# B&R Automation Studio project LW_CapProcess
Automation Studio 4.9

## Configuration Config2

CPU PC_any, AutomationRuntime B4.91, Build 4.1.2, Safety 0.0, Vc V4.73.0

### Task classes (Cpu.sw)
```
Cyclic#1 (cycle 10000 us):
  AlarmsX <- AlarmsPkg.AlarmsX.prg
  CapPush <- CapPushPkg.CapPush.prg
  PickupArm <- PickupArmPkg.PickupArm.prg
  LogoCOnv <- LogoConvPkg.LogoCOnv.prg
  ClrDetect <- ClrDetectPkg.ClrDetect.prg
  LineGates <- LaneGatesPkg.LineGates.prg
  AutoCtrl <- AutoCtrlPkg.AutoCtrl.prg
  SortConv <- SortConvPkg.SortConv.prg
  ComTotal_P <- Libraries.ComTotal.ComTotal_P.prg
DataObjects: Acp10sys
NcDataObjects: acp10etxen <- acp10etxen.dob, gAxis01a <- gAxis01obj.gAxis01a.dob, gAxis01i <- gAxis01obj.gAxis01i.dob, gAxis02a <- gAxis02obj.gAxis02a.dob, gAxis02i <- gAxis02obj.gAxis02i.dob
Binaries: udbdef, mvLoader, arflatprv, TCData, TCLang, arsvcreg, FWRules, arcoal, acp10cfg, Acp10map, iomap, asfw, UserMgt, Alarms, Role, ashwac, sysconf, arconfig, TC, ashwd, User, LogoAxis, Axis01
Libraries: Acp10man, Acp10par, NcGlobal, Acp10sim, Acp10_MC, sys_lib, brsystem, runtime, MpAlarmX, MpBase, astime, MpAxis, MpCom, MpServer, MpUserX, operator, ComTotal_L, AsTCP, standard, ArEventLog, AsBrStr, asieccon, fileio, arcert, dataobj, aseth, ashw, aruser, arssl, powerlnk
```

### Hardware
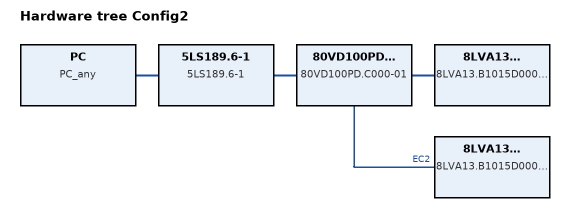
```
5LS189.6-1 : 5LS189.6-1 v1.5.0.0  [SL -> PC.SL1]
80VD100PD.C000-01 : 80VD100PD.C000-01 v2.5.0.0  [PLK1 -> 5LS189.6-1.IF2 (NodeNumber=1) [Cable Type=PowerlinkCable, Length=10, Version=1.0.0.3]; EC1 -> 8LVA13.B1015D000-0.EC; EC2 -> 8LVA13.B1015D000-0a.EC; MT2 -> 8LVA13.B1015D000-0a.MT]
  MotionTP = Acp10Arnc0
  Simulate = standard
  ActiveMotorSimulation_r1 = on
  BothEndSwitchesAreNormallyOpen_r1 = on
  ActiveMotorSimulation_r2 = on
  BothEndSwitchesAreNormallyOpen_r2 = on
8LVA13.B1015D000-0 : 8LVA13.B1015D000-0 v2.2.0.3  [EC -> 80VD100PD.C000-01.EC1; MT -> 80VD100PD.C000-01.MT1]
8LVA13.B1015D000-0a : 8LVA13.B1015D000-0 v2.2.0.3  [EC -> 80VD100PD.C000-01.EC2; MT -> 80VD100PD.C000-01.MT2]
PC : PC_any v1.1.1.0 (OrderNumber=PC)
  ConfigurationID = CapProcess_Config1
  Cyclic1Duration = 10000
  FileDevice1
  FileDeviceName1 = USER
  FileDevicePath1 = USER_PATH
  ActivateOpcUa = 1
  OpcUaInformationModels_PV_Version = 1
```

### Acp10cfg.ncc - PC/Motion/Acp10cfg.ncc
```
NcConfiguration (Version=5.23.1, NcSwId=Acp10)
  ACP10CF1_typ:
    cnt_nettrc_rec_drive = 1500
    bufsize_trace_upload = 1200
    tc_nc_man_task = Cyclic #1
    glob_pv_as_ncobject = Yes
    ncsys_dl_broadcast = Yes
    ncsys_dl_acp_reset = Yes
    safemc_log_err_to_ax = Yes
    network_init:
      ncsw_init_execute = Yes
      automatic_execute = No
      node_nr_warning = Yes
      net_err_before_ncact = Yes
    nettrc:
      enter_parsecrec = Yes
      enter_ncaction = Yes
      save_ring_startidx = Yes
    cam_prof_download:
      cam_dat_dl_parallel = No
      tc_cam_dl_parallel = Task class for NC Manager task
    plk_if[0]:
      if_name = SL1.IF2
      tc_CycDat_PLCopen = Task class for NC Manager task
      mc_broadcast_extdat = No
```

### Acp10map.ncm - PC/Motion/Acp10map.ncm
```
NcMapping (NcSwId=Acp10, DisabledNodesAreHidden=False)
  NcObject gAxis01 (ModuleId=80VD100PD.C000-01, Type=ncAXIS, Channel=1, AcoposSimulation=Standard, InitParameter=gAxis01i, AcoposParameter=gAxis01a, Disabled=FALSE, ModuleDisabled=FALSE)
  NcObject gAxis02 (ModuleId=80VD100PD.C000-01, Type=ncAXIS, Channel=2, AcoposSimulation=Standard, InitParameter=gAxis02i, AcoposParameter=gAxis02a, Disabled=FALSE, ModuleDisabled=FALSE)
  NcObject 80VD100PD.C000-01_ncV_AXIS1 (ModuleId=80VD100PD.C000-01, Type=ncV_AXIS, Channel=1, Disabled=TRUE, ModuleDisabled=FALSE)
  NcObject 80VD100PD.C000-01_ncV_AXIS2 (ModuleId=80VD100PD.C000-01, Type=ncV_AXIS, Channel=2, Disabled=TRUE, ModuleDisabled=FALSE)
```

### LogoAxis.mpaxisbasic - PC/Motion/LogoAxis.mpaxisbasic
```
Element gAxisBasic (Type=mpaxisbasic)
  Alarms = MpAlarmX
```

### SortAxis.mpaxisbasic - PC/Motion/SortAxis.mpaxisbasic
```
Element gAxisBasic_1 (Type=mpaxisbasic)
```

### PvMap.vvm - PC/PvMap.vvm
```iecst
VAR_CONFIG
	::ComTotal_SimInputs.CapPusher_LBK AT %Q.::CapPush:iCapPush.DIs.PusherLBK; (*Insert your comment here...*)
	::ComTotal_SimInputs.LogoAxis_ACTPOS AT %Q.::LogoCOnv:iLogoConv.DIs.LogoActPos; (*Insert your comment here...*)
	::ComTotal_SimInputs.CapPusher_LFR AT %Q.::CapPush:iCapPush.DIs.PusherLFR; (*Insert your comment here...*)
	::ComTotal_SimInputs.MagazineEmpty_IR AT %Q.::CapPush:iCapPush.DIs.MagznPosnEmpty_IR; (*Insert your comment here...*)
	::ComTotal_SimInputs.CapAtPickup_IR AT %Q.::CapPush:iCapPush.DIs.PickUp_IR; (*Insert your comment here...*)
	::ComTotal_SimInputs.ColourDetection_IR AT %Q.::ClrDetect:iClrDetect.DIs.ColorDetectionIR; (*Insert your comment here...*)
	::ComTotal_SimInputs.CapColour_NOT_BLACK AT %Q.::ClrDetect:iClrDetect.DIs.ColorDtectNotBlack; (*Insert your comment here...*)
	::ComTotal_SimInputs.CapColour_METALLIC AT %Q.::ClrDetect:iClrDetect.DIs.ColorDtectMetallic; (*Insert your comment here...*)
	::ComTotal_SimInputs.SortingConveyorStart_IR AT %Q.::SortConv:iSortConv.DIs.SortBasicConvStart_IR; (*Insert your comment here...*)
	::ComTotal_SimInputs.LogoConveyorStart_IR AT %Q.::LogoCOnv:iLogoConv.DIs.LogoConvStart_IR; (*Insert your comment here...*)
	::ComTotal_SimInputs.LogoConveyorExit_IR AT %Q.::LogoCOnv:iLogoConv.DIs.LogoConvExit_IR; (*Insert your comment here...*)
	::ComTotal_SimInputs.LaneGate1_LBK AT %Q.::LineGates:iLineGates.DIs.LG1_LBK; (*Insert your comment here...*)
	::ComTotal_SimInputs.LaneGate1_LFR AT %Q.::LineGates:iLineGates.DIs.LG1_LFR; (*Insert your comment here...*)
	::ComTotal_SimInputs.LaneGate2_LBK AT %Q.::LineGates:iLineGates.DIs.LG2_LBK; (*Insert your comment here...*)
	::ComTotal_SimInputs.LaneGate2_LFR AT %Q.::LineGates:iLineGates.DIs.LG2_LFR; (*Insert your comment here...*)
	::ComTotal_SimInputs.PickupArm_LBK AT %Q.::PickupArm:iPickupArm.DOs.PArmLBK; (*Insert your comment here...*)
	::ComTotal_SimInputs.PickupArm_LFR AT %Q.::PickupArm:iPickupArm.DOs.PArmLFR; (*Insert your comment here...*)
	::ComTotal_SimInputs.CapGripper_VACUUM AT %Q.::PickupArm:iPickupArm.DOs.CapGripVaccum; (*Insert your comment here...*)
	::ComTotal_SimInputs.LaneTop_IR AT %Q.::LineGates:iLineGates.DIs.LaneTopIR; (*Insert your comment here...*)
	::CapPush:iCapPush.DOs.PushFWD AT %Q.::ComTotal_SimOutputs.CapPusher_FWD; (*Insert your comment here...*)
	::SortConv:iSortConv.AOs.SortBasicConvSpeed AT %Q.::ComTotal_SimOutputs.SortingConveyor_SETSPEED; (*Insert your comment here...*)
	::LogoCOnv:iLogoConv.AOs.LogoConvSpeed AT %Q.::ComTotal_SimOutputs.LogoConveyor_SETSPEED; (*Insert your comment here...*)
	::LineGates:iLineGates.DOs.LG1FWD AT %Q.::ComTotal_SimOutputs.LaneGate1_FWD; (*Insert your comment here...*)
	::LineGates:iLineGates.DOs.LW2FWD AT %Q.::ComTotal_SimOutputs.LaneGate2_FWD; (*Insert your comment here...*)
	::PickupArm:iPickupArm.DIs.PArm_FWD AT %Q.::ComTotal_SimOutputs.PickupArm_FWD; (*Insert your comment here...*)
	::PickupArm:iPickupArm.DIs.PArm_BWD AT %Q.::ComTotal_SimOutputs.PickupArm_BWD; (*Insert your comment here...*)
	::PickupArm:iPickupArm.DIs.CapGripper_PICK AT %Q.::ComTotal_SimOutputs.CapGripper_PICK; (*Insert your comment here...*)
	::ClrDetect:iClrDetect.DOs.CapStopperFWD AT %Q.::ComTotal_SimOutputs.CapStopper_FWD; (*Insert your comment here...*)
END_VAR
```

### Alarms.mpalarmxcore - PC/mappServices/Alarms.mpalarmxcore
```
Element gAlarmXCore (Type=mpalarmxcore)
  mapp.AlarmX.Core:
    BySeverity:
      [0]:
        Severity = 50
        [0] = Reaction
          Name = Warning
      [1]:
        Severity = 100
        [0] = Reaction
          Name = EStop
  mapp.AlarmX.Core.Configuration:
    [0]:
      Name = CapPush
      Message = Magzine for cap is empty
      Severity = 10
      Behavior = PersistentAlarm
    [1]:
      Name = PArmError
      Message = Both Arms are on please disable one of it
      Severity = 100
      Behavior = PersistentAlarm
    [2]:
      Name = VaccumError
      Message = Arm is forward but no cap available to pick\
      Severity = 50
      Behavior = PersistentAlarm
    [3]:
      Name = ConvLogoErr
      Message = Cap is on the belt but velocity is zero
      Severity = 100
      Behavior = PersistentAlarm
    [4]:
      Name = ConvSortErr
      Message = Cap is on the belt but velocity is zero
      Severity = 100
      Behavior = PersistentAlarm
    [5]:
      Name = EStopCD
      Message = Estop for Color detect is pressed
      Severity = 100
      Behavior = PersistentAlarm
    [6]:
      Name = CapsFull
      Message = Maximum no of caps are filled please remove
      Severity = 100
      Behavior = PersistentAlarm
    [7]:
      Name = EStopLG
      Message = Emergency stop for line gate
      Severity = 100
      Behavior = PersistentAlarm
    [8]:
      Name = EStopAC
      Message = Emergency stop for main control has been pressed
      Severity = 100
      Behavior = PersistentAlarm
    [9]:
      Name = EStopAuto
      Message = Emergency stop is pressed
      Severity = 100
      Behavior = PersistentAlarm
Element gAlarmXCore_1 (Type=mpalarmxcore)
Element gAlarmXCore_2 (Type=mpalarmxcore)
```

### UserMgt.mpuserx - PC/mappServices/UserMgt.mpuserx
```
Element UserMgmtX (Type=mpuserx)
  ServerSettings:
    Server:
      AdditionalUserData:
        [0] = mail
        [1] = telephoneNumber
  Users:
    DefUser#1:
      id = admin
      lang = en
    DefUser#2:
      id = Anonymous
      lang = en
    DefUser#3:
      id = admin1
      lang = en
    DefUser#4:
      id = dev
      lang = en
    DefUser#5:
      id = yadnesh
      lang = en
  Groups:
    DefGroup#1:
      id = Administrators
      level = 100
      admin = TRUE
    DefGroup#2:
      id = Everyone
      admin = TRUE
    DefGroup#3:
      id = Operator
      level = 80
    DefGroup#4:
      id = Service
      level = 50
```

## Logical view

Binary libraries used (declarations not repeated): operator, runtime, astime, AsIecCon, Acp10man, Acp10par, NcGlobal, Acp10sim 5.23.1, Acp10_MC, sys_lib, brsystem, MpAlarmX, MpBase, MpAxis, MpCom, MpServer, MpUserX, AsTCP, standard, ArEventLog, AsBrStr

### Global.typ - Global data types
```iecst
TYPE
	gMainCmd_Str : 	STRUCT
		Stop : BOOL;
		EStop : BOOL;
		ErrorReset : BOOL;
		Start : BOOL;
	END_STRUCT;
END_TYPE
```

### Global.var - Global variables
```iecst
VAR
	gManuelMode : BOOL;
	gMainCmd : gMainCmd_Str;
	gAxis01 : ACP10AXIS_typ;
	gAxis02 : ACP10AXIS_typ;
	gColorCap : WSTRING[80];
END_VAR
```

### Package Logical/Libraries - Global libraries

### Package Logical/Libraries/ComTotal - Library package for ComTCP

### Library Logical/Libraries/ComTotal/ComTotal_L (ANSIC)

#### MNG_ComHdlr.hpp
```cpp
#ifndef _MNGCOMHDLR_HPP_
#define _MNGCOMHDLR_HPP_

#define TRUE  1
#define FALSE 0

#include "MNG_InternalTyp.hpp"

#include <bur/plc.h>
#include <bur/plctypes.h>
#include <AsTCP.h>
#include <standard.h>
#include <astime.h>
#include <runtime.h>
#include <AsBrStr.h>

typedef struct{
	TcpOpen_typ tcpOpen;
	TcpIoctl_typ tcpIoctl;
	tcpLINGER_typ tcpLINGER;
	TcpSend_typ tcpSend;
	TcpClose_typ tcpClose;
	TcpRecv_typ tcpRecv;
	TcpClient_typ tcpClient;
} asTcpFcn_t;

typedef enum {
	MNG_wSock,
	MNG_skippedMessage
} MNG_errorCases;

typedef enum {
	MNG_Init,
	MNG_Socket,
	MNG_Open,
	MNG_SetIo,
	MNG_Linger,
	MNG_Connecting,
	MNG_Exchange,
	MNG_Closing,
        MNG_Reset
} MNG_internalState_t;

	extern unsigned long int MNG_CpyOutToMsg(MNG_RawDatagram * pToServer, unsigned long int counter, ComTotal_OUTPUTS_32BIT_FWRD *pSimOutputs);
	extern unsigned long int MNG_CpyMsgToInp(MNG_RawDatagram * pFromServer, ComTotal_INPUTS_32BIT_FWRD *pSimInputs);

class MNG_ComHdlr
{
	public:

	MNG_ComHdlr(char *srvIpAdr, unsigned int srvPort, TIME sendCycleTime);
	~MNG_ComHdlr();

        int RunCommunication(void*, void*, BOOL*);

	private:

	char* _srvIpAdr;
	unsigned int _srvPort;
	TIME _sendCycleTime;

	unsigned int _error;

	MNG_internalState_t _internalState;
	TON_typ _connectionTon;
	TIME _connectionTime;

	bool _connect;
	bool _sendDone;

	signed int _recvOffset;

	signed long int _potMsgLen;
	signed long int _totalRecvLen;

	unsigned long int _one;
	unsigned long int _counter;
	unsigned long int _recvLen;
	unsigned long int _recvBuffer[10000];
	TON_typ _sendTon;
	MNG_RawDatagram _recvMessage;
	MNG_RawDatagram _sendMessage;

	static const signed long int SIXTEEN = 16;
	static const unsigned int PORT = 0;
	static const unsigned long int MNG_MAXPAYLOAD = 1400;

	void init_TcpOpen();
	void init_TcpSocket();
	void init_TcpIoctl();
	void init_TcpLinger();
	void init_TcpClient();
	void init_TcpRecv();
	void init_TcpSend(ComTotal_OUTPUTS_32BIT_FWRD* pSimOut);

	void InitParams();

	void SetSendDone(bool toogle);
	void SetStateValue(MNG_internalState_t stateVal);

};
#endif
```

#### MNG_Global.hpp
```cpp
#ifndef  _MNGGLOBAL_HPP_
#define _MNGGLOBAL_HPP_

#include <mng_globalTYP.h>

    typedef struct {

		signed short NumSignals;

        /* BOOL CapPusher_LBK */
        BOOL CapPusher_LBK;
        /* BOOL CapPusher_LFR */
        BOOL CapPusher_LFR;
        /* BOOL MagazineEmpty_IR */
        BOOL MagazineEmpty_IR;
        /* BOOL CapAtPickup_IR */
        BOOL CapAtPickup_IR;
        /* BOOL ColourDetection_IR */
        BOOL ColourDetection_IR;
        /* BOOL CapColour_NOT_BLACK */
        BOOL CapColour_NOT_BLACK;
        /* BOOL CapColour_METALLIC */
        BOOL CapColour_METALLIC;
        /* BOOL SortingConveyorStart_IR */
        BOOL SortingConveyorStart_IR;
        /* BOOL LogoConveyorStart_IR */
        BOOL LogoConveyorStart_IR;
        /* BOOL LogoConveyorExit_IR */
        BOOL LogoConveyorExit_IR;
        /* BOOL LaneGate1_LBK */
        BOOL LaneGate1_LBK;
        /* BOOL LaneGate1_LFR */
        BOOL LaneGate1_LFR;
        /* BOOL LaneGate2_LBK */
        BOOL LaneGate2_LBK;
        /* BOOL LaneGate2_LFR */
        BOOL LaneGate2_LFR;
        /* BOOL PickupArm_LBK */
        BOOL PickupArm_LBK;
        /* BOOL PickupArm_LFR */
        BOOL PickupArm_LFR;
        /* BOOL CapGripper_VACUUM */
        BOOL CapGripper_VACUUM;
        /* BOOL LaneTop_IR */
        BOOL LaneTop_IR;
        /* REAL LogoAxis_ACTPOS */
        REAL LogoAxis_ACTPOS;
        /* BOOL LogoStamper_LBK */
        BOOL LogoStamper_LBK;
        /* BOOL LogoStamper_LFR */
        BOOL LogoStamper_LFR;
        /* REAL PuncherAxis_ACTPOS */
        REAL PuncherAxis_ACTPOS;
        /* BOOL HolePuncher_LBK */
        BOOL HolePuncher_LBK;
        /* BOOL HolePuncher_LFR */
        BOOL HolePuncher_LFR;

        } ComTotal_INPUTS_32BIT_FWRD;

    typedef struct {

		signed short NumSignals;

        /* BOOL CapPusher_FWD */
        BOOL CapPusher_FWD;
        /* REAL SortingConveyor_SETSPEED */
        REAL SortingConveyor_SETSPEED;
        /* BOOL SortingConveyor_CLEAR */
        BOOL SortingConveyor_CLEAR;
        /* REAL LogoConveyor_SETSPEED */
        REAL LogoConveyor_SETSPEED;
        /* BOOL LogoConveyor_CLEAR */
        BOOL LogoConveyor_CLEAR;
        /* BOOL LaneGate1_FWD */
        BOOL LaneGate1_FWD;
        /* BOOL LaneGate2_FWD */
        BOOL LaneGate2_FWD;
        /* BOOL LaneStopper1_CLEAR */
        BOOL LaneStopper1_CLEAR;
        /* BOOL LaneStopper2_CLEAR */
        BOOL LaneStopper2_CLEAR;
        /* BOOL LaneStopper3_CLEAR */
        BOOL LaneStopper3_CLEAR;
        /* BOOL PickupArm_FWD */
        BOOL PickupArm_FWD;
        /* BOOL PickupArm_BWD */
        BOOL PickupArm_BWD;
        /* BOOL CapGripper_PICK */
        BOOL CapGripper_PICK;
        /* BOOL CapStopper_FWD */
        BOOL CapStopper_FWD;
        /* BOOL CP1586_PRESS */
        BOOL CP1586_PRESS;
        /* REAL LogoAxis_SETPOS */
        REAL LogoAxis_SETPOS;
        /* BOOL LogoStamper_FWD */
        BOOL LogoStamper_FWD;
        /* REAL PuncherAxis_SETPOS */
        REAL PuncherAxis_SETPOS;
        /* BOOL HolePuncher_FWD */
        BOOL HolePuncher_FWD;

        } ComTotal_OUTPUTS_32BIT_FWRD;

#endif
```

#### MNG_ComHdlr.cpp
```cpp
#include "MNG_ComHdlr.hpp"
#include "MNG_CpyMsgToInp.cpp"
#include "MNG_CpyOutToMsg.cpp"

asTcpFcn_t _asTcpFcn;

MNG_ComHdlr::MNG_ComHdlr(char *srvIpAdr, unsigned int srvPort, TIME sendCycleTime)
{
	_srvIpAdr = srvIpAdr;
	_srvPort = srvPort;
	_sendCycleTime = sendCycleTime;
	InitParams();
}

MNG_ComHdlr::~MNG_ComHdlr()
{
}

int MNG_ComHdlr::RunCommunication(void* pSimInputs, void* pSimOutputs, BOOL* pSimActive) {

        unsigned long int _lastCounter = _counter;

	ComTotal_INPUTS_32BIT_FWRD* pFwrd_SimInputs = static_cast<ComTotal_INPUTS_32BIT_FWRD*>((pSimInputs));
	ComTotal_OUTPUTS_32BIT_FWRD* pFwrd_SimOutputs = static_cast<ComTotal_OUTPUTS_32BIT_FWRD*>((pSimOutputs));

	switch (_internalState) {

		case MNG_Init:
                        *pSimActive = FALSE;
			_asTcpFcn.tcpOpen.enable = FALSE;
			TcpOpen(&_asTcpFcn.tcpOpen);
			_asTcpFcn.tcpIoctl.enable = FALSE;
			TcpIoctl(&_asTcpFcn.tcpIoctl);
			_asTcpFcn.tcpClient.enable = FALSE;
			TcpClient(&_asTcpFcn.tcpClient);
			_asTcpFcn.tcpSend.enable = FALSE;
			TcpSend(&_asTcpFcn.tcpSend);
			_asTcpFcn.tcpRecv.enable = FALSE;
			TcpRecv(&_asTcpFcn.tcpRecv);
			_asTcpFcn.tcpClose.enable = FALSE;
			TcpClose(&_asTcpFcn.tcpClose);

			_connectionTon.IN = FALSE;
			_connectionTon.PT = _connectionTime;
			_sendTon.IN = FALSE;
			_sendTon.PT = _sendCycleTime;
			SetStateValue(MNG_Socket);
			break;

		case MNG_Socket:
                        *pSimActive = FALSE;
			init_TcpSocket();
			TcpOpen(&_asTcpFcn.tcpOpen);
			_recvOffset = 0;
			if (_connect == 1) {
				SetStateValue(MNG_Open);
				_connectionTon.IN = FALSE;
			}
			break;

		case MNG_Open:
                        *pSimActive = FALSE;
			init_TcpOpen();
			TcpOpen(&_asTcpFcn.tcpOpen);
			if (_asTcpFcn.tcpOpen.status == 0) {
				SetStateValue(MNG_SetIo);
				_asTcpFcn.tcpIoctl.enable = FALSE;
				TcpIoctl(&_asTcpFcn.tcpIoctl);
				_connectionTon.IN = FALSE;
			}
			break;

		case MNG_SetIo:
                        *pSimActive = FALSE;
			init_TcpIoctl();
			TcpIoctl(&_asTcpFcn.tcpIoctl);
			if (_asTcpFcn.tcpIoctl.status == 0) {
				SetStateValue(MNG_Linger);
				_asTcpFcn.tcpClient.enable = FALSE;
				TcpClient(&_asTcpFcn.tcpClient);
				_connectionTon.IN = FALSE;
			}
			break;

		case MNG_Linger:
                        *pSimActive = FALSE;
			init_TcpLinger();
			TcpIoctl(&_asTcpFcn.tcpIoctl);

			if (_asTcpFcn.tcpIoctl.status == 0) {
				SetStateValue(MNG_Connecting);
				_asTcpFcn.tcpClient.enable = FALSE;
				_connectionTon.IN = FALSE;
			}

		case MNG_Connecting:
                        *pSimActive = FALSE;
			_asTcpFcn.tcpClient.enable = TRUE;
			_asTcpFcn.tcpClient.ident = _asTcpFcn.tcpOpen.ident;
			_asTcpFcn.tcpClient.portserv = _srvPort;
			_asTcpFcn.tcpClient.pServer = (long)_srvIpAdr;
			TcpClient(&_asTcpFcn.tcpClient);

			if (_asTcpFcn.tcpClient.status == ERR_FUB_BUSY) {
				// state = state || SetStateValue(Connecting);
			} else if (_asTcpFcn.tcpClient.status == 0) {
				SetStateValue(MNG_Exchange);
				_connectionTon.IN = FALSE;
				SetSendDone(TRUE);
			}
			break;

		case MNG_Exchange:
			init_TcpRecv();
			TcpRecv(&_asTcpFcn.tcpRecv);

			if (_asTcpFcn.tcpRecv.status==0){
                        *pSimActive = FALSE;
			_connectionTon.IN = FALSE;
			_recvLen = _asTcpFcn.tcpRecv.recvlen;
			_potMsgLen = N_TO_HUDINT(_recvBuffer[3]) + SIXTEEN;
			_totalRecvLen = _recvOffset + _recvLen;

			if ((_totalRecvLen < SIXTEEN) || (_totalRecvLen < _potMsgLen)) {
			_recvOffset = _recvOffset + _recvLen;
			}	else {
			while ((_potMsgLen > 0) && (_potMsgLen <= _totalRecvLen)) {
			// misconfigured message sizes
                        if ((unsigned long int)_potMsgLen > sizeof(_recvMessage)) {
			SetStateValue(MNG_Reset);
			break;
			}

			brsmemcpy((unsigned long int) &_recvMessage, (unsigned long int) &_recvBuffer, _potMsgLen*sizeof(unsigned long int));
			_totalRecvLen = _totalRecvLen - _potMsgLen;
			brsmemmove((unsigned long int) &_recvBuffer, (unsigned long int) &_recvBuffer + _potMsgLen, _totalRecvLen*sizeof(unsigned long int));
			_counter = MNG_CpyMsgToInp(&_recvMessage,pFwrd_SimInputs);
                        *pSimActive = (_lastCounter != _counter);
			_recvOffset = _totalRecvLen;

			if (_totalRecvLen > SIXTEEN) {
			_potMsgLen = N_TO_HUDINT(_recvBuffer[3]) + SIXTEEN;
			} else {
			_potMsgLen = 0;
			}

			}
			}
			}

			_sendTon.IN = _sendDone;
			TON(&_sendTon);

			if (_sendTon.Q || _asTcpFcn.tcpSend.enable == 1) {
				if (_sendDone==TRUE) {
					SetSendDone(FALSE);
					MNG_CpyOutToMsg(&_sendMessage, _counter,pFwrd_SimOutputs);
					init_TcpSend(pFwrd_SimOutputs);
				}
				TcpSend(&_asTcpFcn.tcpSend);

				if (_asTcpFcn.tcpSend.status == 0) {
					if (_asTcpFcn.tcpSend.datalen != _asTcpFcn.tcpSend.sentlen) {
						// state = state || SetStateValue(Exchange);
					}
					_asTcpFcn.tcpSend.enable = FALSE;
					SetSendDone(TRUE);
				}
			}
			if (_asTcpFcn.tcpRecv.status == tcpERR_NOT_CONNECTED) {
				SetStateValue(MNG_Closing);
			}
			break;

		case MNG_Closing:
                        *pSimActive = FALSE;
			_asTcpFcn.tcpClose.enable = TRUE;
			_asTcpFcn.tcpClose.ident = _asTcpFcn.tcpOpen.ident;
			_asTcpFcn.tcpClose.how = 0;
			TcpClose(&_asTcpFcn.tcpClose);

			if(_asTcpFcn.tcpClose.status == 0 || _asTcpFcn.tcpClose.status == 32600){
				SetStateValue(MNG_Init);
			}
			break;

                case MNG_Reset:
                        SetStateValue(MNG_Closing);
                        break;
	}

	TON(&_connectionTon);
	_connectionTon.IN = TRUE;
	if (_connectionTon.Q == 1) {
		SetStateValue(MNG_Closing);
		_connectionTon.IN = FALSE;
	}

	return _internalState;
}

void MNG_ComHdlr::init_TcpOpen(){
	_asTcpFcn.tcpOpen.enable = _connect;
}

void MNG_ComHdlr::init_TcpSocket(){
	_asTcpFcn.tcpOpen.enable = TRUE;
	_asTcpFcn.tcpOpen.pIfAddr = 0;
	_asTcpFcn.tcpOpen.port = PORT;
	_asTcpFcn.tcpOpen.options = tcpOPT_REUSEADDR;
}

void MNG_ComHdlr::init_TcpIoctl(){
	_asTcpFcn.tcpIoctl.enable = TRUE;
	_asTcpFcn.tcpIoctl.pData = (unsigned long int) &_one;
	_asTcpFcn.tcpIoctl.datalen = 4;
	_asTcpFcn.tcpIoctl.ident = _asTcpFcn.tcpOpen.ident;
	_asTcpFcn.tcpIoctl.ioctl = tcpTCP_NODELAY_SET;
}

void MNG_ComHdlr::init_TcpLinger(){
	_asTcpFcn.tcpLINGER.lLinger = FALSE;
	_asTcpFcn.tcpLINGER.lOnOff = TRUE;
	_asTcpFcn.tcpIoctl.enable = TRUE;
	_asTcpFcn.tcpIoctl.pData = (unsigned long int) &_asTcpFcn.tcpLINGER;
	_asTcpFcn.tcpIoctl.datalen = sizeof(_asTcpFcn.tcpLINGER);
	_asTcpFcn.tcpIoctl.ident = _asTcpFcn.tcpOpen.ident;
	_asTcpFcn.tcpIoctl.ioctl = tcpSO_LINGER_SET;
}

void MNG_ComHdlr::init_TcpClient(){

	_asTcpFcn.tcpClient.enable = TRUE;
	_asTcpFcn.tcpClient.ident = _asTcpFcn.tcpOpen.ident;
	_asTcpFcn.tcpClient.portserv = _srvPort;
	_asTcpFcn.tcpClient.pServer = (long)_srvIpAdr;
}

void MNG_ComHdlr::init_TcpRecv(){

	_asTcpFcn.tcpRecv.enable = TRUE;
	_asTcpFcn.tcpRecv.ident= _asTcpFcn.tcpOpen.ident;
	_asTcpFcn.tcpRecv.datamax = sizeof(_recvBuffer) - _recvOffset;
	_asTcpFcn.tcpRecv.pData = (unsigned long int) &_recvBuffer + _recvOffset;
}

void MNG_ComHdlr::init_TcpSend(ComTotal_OUTPUTS_32BIT_FWRD *pSimOutputs){

	_asTcpFcn.tcpSend.enable = TRUE;
	_asTcpFcn.tcpSend.ident= _asTcpFcn.tcpOpen.ident;
	_asTcpFcn.tcpSend.datalen = 16 + ((pSimOutputs->NumSignals) + 1) * 4;
	_asTcpFcn.tcpSend.pData = (unsigned long int)&_sendMessage;
	_asTcpFcn.tcpSend.flags = 0;
}

void MNG_ComHdlr::InitParams(){
	_internalState = MNG_Init;
	_connectionTime = 3000;
	_one=1;
	_connect = TRUE;
	_potMsgLen = 0;
	_recvLen = 0;
	_recvOffset = 0;
	_counter = 0;
	SetSendDone(FALSE);
}

void MNG_ComHdlr::SetSendDone(bool toggle){
	_sendDone=toggle;
}

void MNG_ComHdlr::SetStateValue(MNG_internalState_t stateVal){
	_internalState=stateVal;
}
```

#### MNG_CpyMsgToInp.cpp
```cpp
#include "MNG_InternalTyp.hpp"

unsigned long int MNG_CpyMsgToInp(MNG_RawDatagram * pFromServer, ComTotal_INPUTS_32BIT_FWRD *pSimInputs) {

    MNG_DatagramType datagramType;
	unsigned long int DWordBuffer;
        unsigned long int byteCount;
	unsigned long int numSignalsInMessage;

	byteCount = N_TO_HUDINT((pFromServer->Header).ByteCount);
	datagramType = static_cast<MNG_DatagramType>(N_TO_HUDINT((pFromServer->Header).DatagramType));
	if (datagramType != MNG_Raw32BitImage) {
		return 0;
	}

    pSimInputs->NumSignals = 24;

    numSignalsInMessage = N_TO_HUDINT(pFromServer->Payload[0]);
        if ((static_cast<long int>(numSignalsInMessage) != pSimInputs->NumSignals) ||
	(byteCount != 4 + numSignalsInMessage * 4)) {
		return 0;
	}

    /* BOOL CapPusher_LBK */
    pSimInputs->CapPusher_LBK = (pFromServer->Payload[1] != 0);

    /* BOOL CapPusher_LFR */
    pSimInputs->CapPusher_LFR = (pFromServer->Payload[2] != 0);

    /* BOOL MagazineEmpty_IR */
    pSimInputs->MagazineEmpty_IR = (pFromServer->Payload[3] != 0);

    /* BOOL CapAtPickup_IR */
    pSimInputs->CapAtPickup_IR = (pFromServer->Payload[4] != 0);

    /* BOOL ColourDetection_IR */
    pSimInputs->ColourDetection_IR = (pFromServer->Payload[5] != 0);

    /* BOOL CapColour_NOT_BLACK */
    pSimInputs->CapColour_NOT_BLACK = (pFromServer->Payload[6] != 0);

    /* BOOL CapColour_METALLIC */
    pSimInputs->CapColour_METALLIC = (pFromServer->Payload[7] != 0);

    /* BOOL SortingConveyorStart_IR */
    pSimInputs->SortingConveyorStart_IR = (pFromServer->Payload[8] != 0);

    /* BOOL LogoConveyorStart_IR */
    pSimInputs->LogoConveyorStart_IR = (pFromServer->Payload[9] != 0);

    /* BOOL LogoConveyorExit_IR */
    pSimInputs->LogoConveyorExit_IR = (pFromServer->Payload[10] != 0);

    /* BOOL LaneGate1_LBK */
    pSimInputs->LaneGate1_LBK = (pFromServer->Payload[11] != 0);

    /* BOOL LaneGate1_LFR */
    pSimInputs->LaneGate1_LFR = (pFromServer->Payload[12] != 0);

    /* BOOL LaneGate2_LBK */
    pSimInputs->LaneGate2_LBK = (pFromServer->Payload[13] != 0);

    /* BOOL LaneGate2_LFR */
    pSimInputs->LaneGate2_LFR = (pFromServer->Payload[14] != 0);

    /* BOOL PickupArm_LBK */
    pSimInputs->PickupArm_LBK = (pFromServer->Payload[15] != 0);

    /* BOOL PickupArm_LFR */
    pSimInputs->PickupArm_LFR = (pFromServer->Payload[16] != 0);

    /* BOOL CapGripper_VACUUM */
    pSimInputs->CapGripper_VACUUM = (pFromServer->Payload[17] != 0);

    /* BOOL LaneTop_IR */
    pSimInputs->LaneTop_IR = (pFromServer->Payload[18] != 0);

    /* FLOAT32 LogoAxis_ACTPOS */
    DWordBuffer = N_TO_HUDINT(pFromServer->Payload[19]);
    brsmemcpy((unsigned long int)&(pSimInputs->LogoAxis_ACTPOS), (unsigned long int)&(DWordBuffer), 4);

    /* BOOL LogoStamper_LBK */
    pSimInputs->LogoStamper_LBK = (pFromServer->Payload[20] != 0);

    /* BOOL LogoStamper_LFR */
    pSimInputs->LogoStamper_LFR = (pFromServer->Payload[21] != 0);

    /* FLOAT32 PuncherAxis_ACTPOS */
    DWordBuffer = N_TO_HUDINT(pFromServer->Payload[22]);
    brsmemcpy((unsigned long int)&(pSimInputs->PuncherAxis_ACTPOS), (unsigned long int)&(DWordBuffer), 4);

    /* BOOL HolePuncher_LBK */
    pSimInputs->HolePuncher_LBK = (pFromServer->Payload[23] != 0);

    /* BOOL HolePuncher_LFR */
    pSimInputs->HolePuncher_LFR = (pFromServer->Payload[24] != 0);

return N_TO_HUDINT((pFromServer->Header).Counter); // return counter
}
```

#### MNG_CpyOutToMsg.cpp
```cpp
#include "MNG_InternalTyp.hpp"

unsigned long int MNG_CpyOutToMsg(MNG_RawDatagram * pToServer, unsigned long int counter, ComTotal_OUTPUTS_32BIT_FWRD *pSimOutputs ) {

        unsigned long int DWordBuffer;

        pSimOutputs->NumSignals = 19;
        (pToServer->Header).ByteCount    = H_TO_NUDINT(80);
        (pToServer->Header).DatagramType = H_TO_NUDINT(MNG_Raw32BitImage);
        (pToServer->Header).SentTime = H_TO_NUDINT(0);  // Todo
        (pToServer->Header).Counter = H_TO_NUDINT(counter);
        pToServer->Payload[0] = H_TO_NUDINT(pSimOutputs->NumSignals);

    /* CapPusher_FWD : BOOL */
    if(pSimOutputs->CapPusher_FWD == 1) {
        pToServer->Payload[1] = 0xFFFFFFFF;   /*BOOL */
    } else {
        pToServer->Payload[1] = 0;
    }

    /* SortingConveyor_SETSPEED : FLOAT32 */
    brsmemcpy((unsigned long int)&(DWordBuffer), (unsigned long int)&(pSimOutputs->SortingConveyor_SETSPEED), 4);
    pToServer->Payload[2] = H_TO_NUDINT(DWordBuffer);

    /* SortingConveyor_CLEAR : BOOL */
    if(pSimOutputs->SortingConveyor_CLEAR == 1) {
        pToServer->Payload[3] = 0xFFFFFFFF;   /*BOOL */
    } else {
        pToServer->Payload[3] = 0;
    }

    /* LogoConveyor_SETSPEED : FLOAT32 */
    brsmemcpy((unsigned long int)&(DWordBuffer), (unsigned long int)&(pSimOutputs->LogoConveyor_SETSPEED), 4);
    pToServer->Payload[4] = H_TO_NUDINT(DWordBuffer);

    /* LogoConveyor_CLEAR : BOOL */
    if(pSimOutputs->LogoConveyor_CLEAR == 1) {
        pToServer->Payload[5] = 0xFFFFFFFF;   /*BOOL */
    } else {
        pToServer->Payload[5] = 0;
    }

    /* LaneGate1_FWD : BOOL */
    if(pSimOutputs->LaneGate1_FWD == 1) {
        pToServer->Payload[6] = 0xFFFFFFFF;   /*BOOL */
    } else {
        pToServer->Payload[6] = 0;
    }

    /* LaneGate2_FWD : BOOL */
    if(pSimOutputs->LaneGate2_FWD == 1) {
        pToServer->Payload[7] = 0xFFFFFFFF;   /*BOOL */
    } else {
        pToServer->Payload[7] = 0;
    }

    /* LaneStopper1_CLEAR : BOOL */
    if(pSimOutputs->LaneStopper1_CLEAR == 1) {
        pToServer->Payload[8] = 0xFFFFFFFF;   /*BOOL */
    } else {
        pToServer->Payload[8] = 0;
    }

    /* LaneStopper2_CLEAR : BOOL */
    if(pSimOutputs->LaneStopper2_CLEAR == 1) {
        pToServer->Payload[9] = 0xFFFFFFFF;   /*BOOL */
    } else {
        pToServer->Payload[9] = 0;
    }

    /* LaneStopper3_CLEAR : BOOL */
    if(pSimOutputs->LaneStopper3_CLEAR == 1) {
        pToServer->Payload[10] = 0xFFFFFFFF;   /*BOOL */
    } else {
        pToServer->Payload[10] = 0;
    }

    /* PickupArm_FWD : BOOL */
    if(pSimOutputs->PickupArm_FWD == 1) {
        pToServer->Payload[11] = 0xFFFFFFFF;   /*BOOL */
    } else {
        pToServer->Payload[11] = 0;
    }

    /* PickupArm_BWD : BOOL */
    if(pSimOutputs->PickupArm_BWD == 1) {
        pToServer->Payload[12] = 0xFFFFFFFF;   /*BOOL */
    } else {
        pToServer->Payload[12] = 0;
    }

    /* CapGripper_PICK : BOOL */
    if(pSimOutputs->CapGripper_PICK == 1) {
        pToServer->Payload[13] = 0xFFFFFFFF;   /*BOOL */
    } else {
        pToServer->Payload[13] = 0;
    }

    /* CapStopper_FWD : BOOL */
    if(pSimOutputs->CapStopper_FWD == 1) {
        pToServer->Payload[14] = 0xFFFFFFFF;   /*BOOL */
    } else {
        pToServer->Payload[14] = 0;
    }

    /* CP1586_PRESS : BOOL */
    if(pSimOutputs->CP1586_PRESS == 1) {
        pToServer->Payload[15] = 0xFFFFFFFF;   /*BOOL */
    } else {
        pToServer->Payload[15] = 0;
    }

    /* LogoAxis_SETPOS : FLOAT32 */
    brsmemcpy((unsigned long int)&(DWordBuffer), (unsigned long int)&(pSimOutputs->LogoAxis_SETPOS), 4);
    pToServer->Payload[16] = H_TO_NUDINT(DWordBuffer);

    /* LogoStamper_FWD : BOOL */
    if(pSimOutputs->LogoStamper_FWD == 1) {
        pToServer->Payload[17] = 0xFFFFFFFF;   /*BOOL */
    } else {
        pToServer->Payload[17] = 0;
    }

    /* PuncherAxis_SETPOS : FLOAT32 */
    brsmemcpy((unsigned long int)&(DWordBuffer), (unsigned long int)&(pSimOutputs->PuncherAxis_SETPOS), 4);
    pToServer->Payload[18] = H_TO_NUDINT(DWordBuffer);

    /* HolePuncher_FWD : BOOL */
    if(pSimOutputs->HolePuncher_FWD == 1) {
        pToServer->Payload[19] = 0xFFFFFFFF;   /*BOOL */
    } else {
        pToServer->Payload[19] = 0;
    }

	return 0;
}
```

### Program Logical/Libraries/ComTotal/ComTotal_P (ANSIC)

#### Main.cpp
```cpp
#include <bur/plctypes.h>

#include "../ComTotal_L/MNG_Global.hpp"
#include "../ComTotal_L/MNG_InternalTyp.hpp"
#include "../ComTotal_L/MNG_ComHdlr.hpp"

#include <MNG_PackageTyp.h>
#include <MNG_PackageVAR.h>
#include <TypesTYP.h>
#include <VariablesVAR.h>

unsigned long bur_heap_size = 0x4FFFF;

MNG_ComHdlr *pMNG_ComHdlr;

void _INIT ProgramInit(void)
{
    pMNG_ComHdlr = new MNG_ComHdlr(ComTotal_SimServerAddress, ComTotal_SimServerPort, ComTotal_SimSendCycleTime);
}

void _CYCLIC ProgramCyclic(void)
{
    connectionState = pMNG_ComHdlr->RunCommunication((void*)&ComTotal_SimInputs,(void*)&ComTotal_SimOutputs, &ComTotal_SimActive);
}

void _EXIT ProgramExit(void)
{
    delete pMNG_ComHdlr;
}
```

### MNG_Package.typ
```iecst
(*                                                                            *)
(* File generated by the B&R AS 4 control config generator                    *)
(*                                                                            *)
(*     Provider: machineering                                                 *)
(*  Application: iPhysics_2.4.master                                          *)
(* Architecture: Windows 64 Bit                                               *)
(*      Version: 2.4.12706.master                                             *)
(*        Build: 608a88cb4                                                    *)
(*         Date: 2022-07-25, Time: 11:40:12                                   *)
(*                                                                            *)

TYPE
ComTotal_INPUTS_32BIT : STRUCT

		NumSignals	: INT := 24;

        CapPusher_LBK : BOOL := 0;
        (* BOOL CapPusher_LBK *)
        CapPusher_LFR : BOOL := 0;
        (* BOOL CapPusher_LFR *)
        MagazineEmpty_IR : BOOL := 0;
        (* BOOL MagazineEmpty_IR *)
        CapAtPickup_IR : BOOL := 0;
        (* BOOL CapAtPickup_IR *)
        ColourDetection_IR : BOOL := 0;
        (* BOOL ColourDetection_IR *)
        CapColour_NOT_BLACK : BOOL := 0;
        (* BOOL CapColour_NOT_BLACK *)
        CapColour_METALLIC : BOOL := 0;
        (* BOOL CapColour_METALLIC *)
        SortingConveyorStart_IR : BOOL := 0;
        (* BOOL SortingConveyorStart_IR *)
        LogoConveyorStart_IR : BOOL := 0;
        (* BOOL LogoConveyorStart_IR *)
        LogoConveyorExit_IR : BOOL := 0;
        (* BOOL LogoConveyorExit_IR *)
        LaneGate1_LBK : BOOL := 0;
        (* BOOL LaneGate1_LBK *)
        LaneGate1_LFR : BOOL := 0;
        (* BOOL LaneGate1_LFR *)
        LaneGate2_LBK : BOOL := 0;
        (* BOOL LaneGate2_LBK *)
        LaneGate2_LFR : BOOL := 0;
        (* BOOL LaneGate2_LFR *)
        PickupArm_LBK : BOOL := 0;
        (* BOOL PickupArm_LBK *)
        PickupArm_LFR : BOOL := 0;
        (* BOOL PickupArm_LFR *)
        CapGripper_VACUUM : BOOL := 0;
        (* BOOL CapGripper_VACUUM *)
        LaneTop_IR : BOOL := 0;
        (* BOOL LaneTop_IR *)
        LogoAxis_ACTPOS : REAL := 0.0;
        (* REAL LogoAxis_ACTPOS *)
        LogoStamper_LBK : BOOL := 0;
        (* BOOL LogoStamper_LBK *)
        LogoStamper_LFR : BOOL := 0;
        (* BOOL LogoStamper_LFR *)
        PuncherAxis_ACTPOS : REAL := 0.0;
        (* REAL PuncherAxis_ACTPOS *)
        HolePuncher_LBK : BOOL := 0;
        (* BOOL HolePuncher_LBK *)
        HolePuncher_LFR : BOOL := 0;
        (* BOOL HolePuncher_LFR *)

	END_STRUCT;

ComTotal_OUTPUTS_32BIT : STRUCT

		NumSignals	: INT := 19;

        CapPusher_FWD : BOOL := 0;
        (* BOOL CapPusher_FWD *)
        SortingConveyor_SETSPEED : REAL := 0.0;
        (* REAL SortingConveyor_SETSPEED *)
        SortingConveyor_CLEAR : BOOL := 0;
        (* BOOL SortingConveyor_CLEAR *)
        LogoConveyor_SETSPEED : REAL := 0.0;
        (* REAL LogoConveyor_SETSPEED *)
        LogoConveyor_CLEAR : BOOL := 0;
        (* BOOL LogoConveyor_CLEAR *)
        LaneGate1_FWD : BOOL := 0;
        (* BOOL LaneGate1_FWD *)
        LaneGate2_FWD : BOOL := 0;
        (* BOOL LaneGate2_FWD *)
        LaneStopper1_CLEAR : BOOL := 0;
        (* BOOL LaneStopper1_CLEAR *)
        LaneStopper2_CLEAR : BOOL := 0;
        (* BOOL LaneStopper2_CLEAR *)
        LaneStopper3_CLEAR : BOOL := 0;
        (* BOOL LaneStopper3_CLEAR *)
        PickupArm_FWD : BOOL := 0;
        (* BOOL PickupArm_FWD *)
        PickupArm_BWD : BOOL := 0;
        (* BOOL PickupArm_BWD *)
        CapGripper_PICK : BOOL := 0;
        (* BOOL CapGripper_PICK *)
        CapStopper_FWD : BOOL := 0;
        (* BOOL CapStopper_FWD *)
        CP1586_PRESS : BOOL := 0;
        (* BOOL CP1586_PRESS *)
        LogoAxis_SETPOS : REAL := 0.0;
        (* REAL LogoAxis_SETPOS *)
        LogoStamper_FWD : BOOL := 0;
        (* BOOL LogoStamper_FWD *)
        PuncherAxis_SETPOS : REAL := 0.0;
        (* REAL PuncherAxis_SETPOS *)
        HolePuncher_FWD : BOOL := 0;
        (* BOOL HolePuncher_FWD *)

	END_STRUCT;

END_TYPE
```

### MNG_Package.var
```iecst
(*                                                                            *)
(* File generated by the B&R AS 4 control config generator                    *)
(*                                                                            *)
(*     Provider: machineering                                                 *)
(*  Application: iPhysics_2.4.master                                          *)
(* Architecture: Windows 64 Bit                                               *)
(*      Version: 2.4.12706.master                                             *)
(*        Build: 608a88cb4                                                    *)
(*         Date: 2022-07-25, Time: 11:40:12                                   *)
(*                                                                            *)
VAR
	ComTotal_SimInputs : ComTotal_INPUTS_32BIT := (0);
	ComTotal_SimOutputs : ComTotal_OUTPUTS_32BIT := (0);
	ComTotal_SimServerAddress : STRING[15] := '127.0.0.1';
	ComTotal_SimServerPort : UINT := 5000;
	ComTotal_SimSendCycleTime : TIME := T#5ms;
	ComTotal_SimActive : BOOL := FALSE;
END_VAR
```

### Package Logical/gAxis01obj - gAxis01obj

### gAxis01i.ax
```
InitParameter (Version=5.23.1, NcSwId=Acp10)
  ACP10AXIS_typ:
    dig_in:
      level:
        reference = ncACTIV_HI
        pos_hw_end = ncACTIV_HI
        neg_hw_end = ncACTIV_HI
        trigger1 = ncACTIV_HI
        trigger2 = ncACTIV_LO + ncQUICKSTOP
    encoder_if:
      parameter:
        count_dir = ncSTANDARD
        scaling:
          load:
            units = 7000
            rev_motor = 1
    limit:
      parameter:
        v_pos = 10000
        v_neg = 10000
        a1_pos = 50000
        a2_pos = 50000
        a1_neg = 50000
        a2_neg = 50000
        t_jolt = 0
        t_in_pos = 0
        pos_sw_end = 2000000000
        neg_sw_end = -2000000000
        ds_warning = 500
        ds_stop = 1000
        a_stop = 1.0e30
        dv_stop = 0
        dv_stop_mode = ncOFF
    controller:
      mode = ncPOSITION
      position:
        kv = 50
        tn = 0
        t_predict = 0.0004
        t_total = 0.0004
        p_max = 1.0e30
        i_max = 0
      speed:
        kv = 2.0
        tn = 0
        t_filter = 0.0
        isq_filter1:
          type = ncOFF
          a0 = 0.0
          a1 = 0.0
          b0 = 0.0
          b1 = 0.0
          b2 = 0.0
          c0_par_id = 0
          c1_par_id = 0
        isq_filter2:
          type = ncOFF
          a0 = 0.0
          a1 = 0.0
          b0 = 0.0
          b1 = 0.0
          b2 = 0.0
          c0_par_id = 0
          c1_par_id = 0
        isq_filter3:
          type = ncOFF
          a0 = 0.0
          a1 = 0.0
          b0 = 0.0
          b1 = 0.0
          b2 = 0.0
          c0_par_id = 0
          c1_par_id = 0
      uf:
        type = ncLINEAR + ncCORRECTION
        auto_config = ncMOTOR_PAR
        u0 = 0
        un = 0
        fn = 50.0
        k_f_slip = 0
      ff:
        mode = ncSTANDARD
        torque_load = 0.0
        torque_pos = 0.0
        torque_neg = 0.0
        kv_torque = 0.0
        inertia = 0.0
        t_filter_a = 0.0
      fb:
        mode = ncSTANDARD
        speed_mix_ratio = 0.0
        speed_kv = 2.0
      model:
        mass1:
          inertia = 0
          viscous_friction = 0
        mass2:
          inertia = 0
          viscous_friction = 0
          stiffness = 0
          damping = 0
    move:
      stop:
        parameter[0]:
          decel_ramp = ncA_LIMIT
          controller = ncON
        parameter[1]:
          decel_ramp = ncA_LIMIT
          controller = ncON
        parameter[2]:
          decel_ramp = ncA_LIMIT
          controller = ncON
        parameter[3]:
          decel_ramp = ncA_LIMIT
          controller = ncON
        quickstop:
          decel_ramp = ncA_LIMIT
          t_jolt = 0
        drive_error:
          decel_ramp = ncA_LIMIT
      homing:
        parameter:
          s = 0
          v_switch = 5000
          v_trigger = 500
          a = 50000
          mode = ncDIRECT
          edge_sw = ncPOSITIVE
          start_dir = ncPOSITIVE
          trigg_dir = ncPOSITIVE
          ref_pulse = ncOFF
          fix_dir = ncOFF
          tr_s_block = 0
          torque_lim = 0
          ds_block = 0
          ds_stop = 0
      basis:
        parameter:
          v_pos = 5000
          v_neg = 5000
          a1_pos = 50000
          a2_pos = 50000
          a1_neg = 50000
          a2_neg = 50000
    message:
      text:
        parameter:
          format = ncBREAK
          columns = 80
          data_modul = acp10etxen
```

### Package Logical/gAxis02obj - gAxis02obj

### gAxis02i.ax
```
InitParameter (Version=5.23.1, NcSwId=Acp10)
  ACP10AXIS_typ:
    dig_in:
      level:
        reference = ncACTIV_HI
        pos_hw_end = ncACTIV_HI
        neg_hw_end = ncACTIV_HI
        trigger1 = ncACTIV_HI
        trigger2 = ncACTIV_LO + ncQUICKSTOP
    encoder_if:
      parameter:
        count_dir = ncSTANDARD
        scaling:
          load:
            units = 7000
            rev_motor = 1
    limit:
      parameter:
        v_pos = 25000.0
        v_neg = 25000.0
        a1_pos = 250000.0
        a2_pos = 250000.0
        a1_neg = 250000.0
        a2_neg = 250000.0
        t_jolt = 0.123
        t_in_pos = 0.123
        pos_sw_end = 2000000000
        neg_sw_end = -2000000000
        ds_warning = 350.0
        ds_stop = 700.0
        a_stop = 1.0e30
        dv_stop = 0
        dv_stop_mode = ncOFF
    controller:
      mode = ncPOSITION
      position:
        kv = 50
        tn = 0
        t_predict = 0.0004
        t_total = 0.0004
        p_max = 1.0e30
        i_max = 0
      speed:
        kv = 2.0
        tn = 0
        t_filter = 0.0
        isq_filter1:
          type = ncOFF
          a0 = 0.0
          a1 = 0.0
          b0 = 0.0
          b1 = 0.0
          b2 = 0.0
          c0_par_id = 0
          c1_par_id = 0
        isq_filter2:
          type = ncOFF
          a0 = 0.0
          a1 = 0.0
          b0 = 0.0
          b1 = 0.0
          b2 = 0.0
          c0_par_id = 0
          c1_par_id = 0
        isq_filter3:
          type = ncOFF
          a0 = 0.0
          a1 = 0.0
          b0 = 0.0
          b1 = 0.0
          b2 = 0.0
          c0_par_id = 0
          c1_par_id = 0
      uf:
        type = ncLINEAR + ncCORRECTION
        auto_config = ncMOTOR_PAR
        u0 = 0
        un = 0
        fn = 50.0
        k_f_slip = 0
      ff:
        mode = ncSTANDARD
        torque_load = 0.0
        torque_pos = 0.0
        torque_neg = 0.0
        kv_torque = 0.0
        inertia = 0.0
        t_filter_a = 0.0
      fb:
        mode = ncSTANDARD
        speed_mix_ratio = 0.0
        speed_kv = 2.0
      model:
        mass1:
          inertia = 0
          viscous_friction = 0
        mass2:
          inertia = 0
          viscous_friction = 0
          stiffness = 0
          damping = 0
    move:
      stop:
        parameter[0]:
          decel_ramp = ncA_LIMIT
          controller = ncON
        parameter[1]:
          decel_ramp = ncA_LIMIT
          controller = ncON
        parameter[2]:
          decel_ramp = ncA_LIMIT
          controller = ncON
        parameter[3]:
          decel_ramp = ncA_LIMIT
          controller = ncON
        quickstop:
          decel_ramp = ncA_LIMIT
          t_jolt = 0
        drive_error:
          decel_ramp = ncA_LIMIT
      homing:
        parameter:
          s = 0
          v_switch = 5000
          v_trigger = 500
          a = 50000
          mode = ncDIRECT
          edge_sw = ncPOSITIVE
          start_dir = ncPOSITIVE
          trigg_dir = ncPOSITIVE
          ref_pulse = ncOFF
          fix_dir = ncOFF
          tr_s_block = 0
          torque_lim = 0
          ds_block = 0
          ds_stop = 0
      basis:
        parameter:
          v_pos = 5000
          v_neg = 5000
          a1_pos = 50000
          a2_pos = 50000
          a1_neg = 50000
          a2_neg = 50000
    message:
      text:
        parameter:
          format = ncBREAK
          columns = 80
          data_modul = acp10etxen
```

### Program Logical/AlarmsPkg/AlarmsX

#### Variables.var
```iecst
VAR
	MpAlarmXHistory_0 : MpAlarmXHistory;
	MpAlarmXHistoryUI_0 : MpAlarmXHistoryUI;
	UiConnectHostory : MpAlarmXHistoryUIConnectType := (0); (*String which defines language and unit for display and export*)
	iFb_AlarmX : MpAlarmXCore;
	iFb_AlarmUI : MpAlarmXListUI;
	UIConnectCore : MpAlarmXListUIConnectType;
END_VAR
```

#### Main.st
```iecst
(*|ŻŻŻŻŻŻŻŻŻŻŻŻŻŻŻŻŻŻŻŻŻŻŻŻŻŻŻŻŻŻŻŻŻŻŻŻŻŻŻŻŻŻŻŻŻŻŻŻŻŻŻŻŻŻŻŻŻŻŻŻŻŻŻŻŻŻŻŻŻŻŻŻŻŻŻŻŻŻŻŻŻŻŻŻŻŻŻŻŻŻŻŻŻŻŻŻŻŻŻŻŻŻŻŻŻŻŻŻŻŻ|*)
(*| Copyright      :-  B&R Industrial Automation GmbH															 |*)
(*| Contact Person :-  maskeu																					 |*)
(*|——————————————————————————————————————————————————————————————————————————————————————————————————————————————|*)
(*| System       :-  TODO: Sewing Machine                                                                        |*)
(*| Task Name    :-  TODO: Dosctrl                                                                   	         |*)
(*| Auther Name  :-  maskeu																						 |*)
(*| Created Date :-  October 10, 2023 																		   	 |*)
(*| Task Class   :-  Task Class #1                                                                               |*)
(*| Task Time    :-  Task Timing 10mSec                                                                          |*)
(*| OS Version   :-  V0.00.0                                                                                     |*)
(*| AS Version   :-  AS 4.12.4.107                                                                               |*)
(*|——————————————————————————————————————————————————————————————————————————————————————————————————————————————|*)
(*| Description  :-  Dosing Control                                                            |*)
(*|                                                                                                              |*)
(*|——————————————————————————————————————————————————————————————————————————————————————————————————————————————|*)
(*| History (Task Modification):                                                                                 |*)
(*|                                                                                                              |*)
(*| Version      Date       Modified By      Modification                                             Status     |*)
(*| V1.00.0   10/10/2023    maskeu        TODO: Insert Modification Done                       Update Status     |*)
(*|______________________________________________________________________________________________________________|*)

PROGRAM _INIT
	(* Insert code here *)

END_PROGRAM

PROGRAM _CYCLIC
	(* Insert code here *)
	// alarmx on
	iFb_AlarmX.Enable:=TRUE;
	iFb_AlarmX.MpLink:=ADR(gAlarmXCore);

	iFb_AlarmUI.Enable:=TRUE;
	iFb_AlarmUI.MpLink:=ADR(gAlarmXCore);
	iFb_AlarmUI.UIConnect:=ADR(UIConnectCore);

	iFb_AlarmX();
	iFb_AlarmUI();

END_PROGRAM

PROGRAM _EXIT
	(* Insert code here *)

	iFb_AlarmUI.Enable:=FALSE;
	iFb_AlarmX.Enable:=FALSE;
	iFb_AlarmX();
	iFb_AlarmUI();
END_PROGRAM
```

### Program Logical/CapPushPkg/CapPush (IEC)

#### Main.st - Init, cyclic, exit code
```iecst
PROGRAM _INIT
END_PROGRAM

PROGRAM _CYCLIC

	CASE sCapPushStep OF

		//wait state if statred will move in next state
		enWAIT:
		//	iCapPush.DOs.PushFWD:=FALSE;
			iCapPush.Status.Running:=FALSE;
			IF iCapPush.Cmd.Start=TRUE THEN
				iCapPush.Cmd.Start:=FALSE;
				sCapPushStep:=enPUSH;
			END_IF;

			//pushing the cap
		enPUSH:
			iCapPush.Status.Running:=TRUE;
			IF iCapPush.DIs.MagznPosnEmpty_IR=FALSE AND iCapPush.DIs.PickUp_IR=FALSE THEN
				iCapPush.DOs.PushFWD:=TRUE ;
				sCapPushStep:=enOPERATION;
			END_IF;

			//OPERATION Mode
		enOPERATION:
			IF iCapPush.DOs.PushFWD=FALSE  THEN
				sCapPushStep:=enWAIT;

			END_IF;
			sCapPushStep:=enWAIT;

			//error mode
		enERROR:
			iCapPush.DOs.PushFWD:=FALSE ;
			iCapPush.Cmd.Start:=FALSE;
			IF  iCapPush.Cmd.ErrorReset=TRUE THEN
				iCapPush.Cmd.ErrorReset:=TRUE ;
				sCapPushStep:=enWAIT;
			END_IF;

	END_CASE;
END_PROGRAM

PROGRAM _EXIT

END_PROGRAM
```

#### Types.typ - Local data types
```iecst
TYPE
	sStep_CapPush :
		(
		enWAIT,
		enPUSH,
		enOPERATION,
		enERROR
		);
END_TYPE
```

#### Variables.var - Local variables
```iecst
VAR
	iCapPush : CapPush_typ;
END_VAR
VAR RETAIN
	sCapPushStep : sStep_CapPush;
END_VAR
```

#### AlarmsCP.st
```iecst
ACTION AlarmsCP:

	IF iCapPush.DIs.MagznPosnEmpty_IR=TRUE THEN
		MpAlarmXSet(gAlarmXCore, 'CapPush');
		IF MpAlarmXCheckReaction(gAlarmXCore, 'Warning') THEN
		//	iCapPush.Status.Error:=TRUE ;
	//		iCapPush.DOs.PushFWD:=TRUE;
		END_IF
	ELSE
		MpAlarmXReset(gAlarmXCore, 'CapPush');
	END_IF

END_ACTION
```

### CapPushtyp.typ
```iecst
TYPE
	CmdCapPush_typ : 	STRUCT
		Start : BOOL;
		Estop : BOOL;
		Stop : BOOL;
		ErrorReset : BOOL;
	END_STRUCT;
	CapPush_typ : 	STRUCT
		Cmd : CmdCapPush_typ;
		DIs : CapPushDIs_typ;
		DOs : CapPushDOs_typ;
		Status : StatusCapPush_typ;
	END_STRUCT;
	StatusCapPush_typ : 	STRUCT
		Pushing : BOOL;
		Running : BOOL;
		Backing : BOOL;
		Error : BOOL;
	END_STRUCT;
	CapPushDIs_typ : 	STRUCT
		PusherLBK : BOOL;
		PusherLFR : BOOL;
		PickUp_IR : BOOL;
		MagznPosnEmpty_IR : BOOL;
	END_STRUCT;
	CapPushDOs_typ : 	STRUCT
		PushFWD : BOOL;
	END_STRUCT;
END_TYPE
```

### Program Logical/PickupArmPkg/PickupArm (IEC)

#### Main.st - Init, cyclic, exit code
```iecst
PROGRAM _INIT
	(* Insert code here *)

END_PROGRAM

PROGRAM _CYCLIC
	(* Insert code here *)

	CASE sPArmStep OF

		//wait state
		enWAIT:

			iPickupArm.DIs.PArm_FWD:=FALSE;
			iPickupArm.DIs.PArm_BWD:=FALSE;
			IF iPickupArm.Cmd.Start=TRUE THEN
				iPickupArm.Cmd.Start:=FALSE;
				sPArmStep:=enPICKING;
			END_IF;

			//picking the caps
		enPICKING:

			iPickupArm.DIs.PArm_FWD:=TRUE;
			IF iPickupArm.DOs.PArmLFR = TRUE THEN
				IF gManuelMode=TRUE THEN

				ELSE
					iPickupArm.DIs.CapGripper_PICK:=TRUE;
				END_IF;
			END_IF;
			IF iPickupArm.DOs.CapGripVaccum=TRUE THEN
				iPickupArm.DIs.PArm_FWD:=FALSE;
				sPArmStep:=enDROPPING;
			END_IF;

			//dropping caps on conveyor
		enDROPPING:
			iPickupArm.DIs.PArm_BWD:=TRUE;
			IF iPickupArm.DOs.PArmLBK=TRUE THEN
				iPickupArm.DIs.PArm_BWD:=FALSE;
				IF gManuelMode=TRUE THEN

				ELSE
					iPickupArm.DIs.CapGripper_PICK:=FALSE;
				END_IF;
				IF iPickupArm.DIs.CapGripper_PICK=FALSE THEN
					sPArmStep:=enWAIT;
				END_IF;
			END_IF;

			//error mode
		enERROR:
			iPickupArm.DIs.PArm_FWD:=FALSE;
			iPickupArm.DIs.PArm_BWD:=TRUE;
			IF iPickupArm.DOs.PArmLBK=TRUE THEN
				iPickupArm.DIs.PArm_BWD:=FALSE;
				iPickupArm.DIs.CapGripper_PICK:=FALSE;
			END_IF;
			IF iPickupArm.Cmd.ErrorReset=TRUE THEN
				iPickupArm.Cmd.ErrorReset:=FALSE;
				sPArmStep:=enWAIT;
			END_IF;
	END_CASE;
END_PROGRAM

PROGRAM _EXIT
	(* Insert code here *)

END_PROGRAM
```

#### Types.typ - Local data types
```iecst
TYPE
	sStep_PArm :
		(
		enWAIT,
		enPICKING,
		enDROPPING,
		enOPERATION,
		enERROR
		);
END_TYPE
```

#### Variables.var - Local variables
```iecst
VAR
	iPickupArm : PickupArm_typ;
END_VAR
VAR RETAIN
	sPArmStep : sStep_PArm;
END_VAR
```

#### AlarmsPA.st
```iecst
ACTION AlarmsPA:

	IF  iPickupArm.DIs.PArm_BWD=TRUE AND iPickupArm.DIs.PArm_FWD=TRUE THEN
		MpAlarmXSet(gAlarmXCore, 'PArmError');
		IF MpAlarmXCheckReaction(gAlarmXCore, 'EStop') THEN
			//	iCapPush.Status.Error:=TRUE ;
		END_IF
	ELSE
		MpAlarmXReset(gAlarmXCore, 'PArmError');
	END_IF

	IF iPickupArm.DOs.PArmLFR =TRUE AND iPickupArm.DOs.CapGripVaccum=FALSE THEN
		MpAlarmXSet(gAlarmXCore, 'VaccumError');
		IF MpAlarmXCheckReaction(gAlarmXCore, 'Warning') THEN
			//	iCapPush.Status.Error:=TRUE ;
		END_IF
	ELSE
		MpAlarmXReset(gAlarmXCore, 'VaccumError');
	END_IF
END_ACTION
```

### Pickuptyp.typ
```iecst
(*Main control for pickup arm*)

TYPE
	PickupArm_typ : 	STRUCT
		DOs : DOs_typ; (*digital outputs*)
		Cmd : PArmCmd_typ; (*commands*)
		Status : PArmStatus_typ; (*status of arm*)
		DIs : DIs_typ; (*digital inputs*)
	END_STRUCT;
END_TYPE

(*pickuparm status*)

TYPE
	PArmStatus_typ : 	STRUCT  (*status of arm*)
		Running : BOOL; (*running*)
		PickingUp : BOOL; (*picking up cap*)
		Dropping : BOOL; (*dropping cap*)
		Holding : BOOL; (*holding cap*)
		Error : BOOL; (*error mode*)
	END_STRUCT;
END_TYPE

(*commands for parm*)

TYPE
	PArmCmd_typ : 	STRUCT  (*command strcture*)
		Start : BOOL; (*starting the arm*)
		Stop : BOOL; (*stopping the arm'*)
		Estop : BOOL; (*emergency stopping arm*)
		ErrorReset : BOOL;
	END_STRUCT;
END_TYPE

(*digital outputs*)

TYPE
	DOs_typ : 	STRUCT  (*digital outputs structure*)
		PArmLFR : BOOL; (*parm left forewarding*)
		PArmLBK : BOOL; (*arm left backword*)
		CapGripVaccum : BOOL; (*cap gripping by vaccume*)
	END_STRUCT;
END_TYPE

(*digital inputs*)

TYPE
	DIs_typ : 	STRUCT
		PArm_FWD : BOOL; (*arm going forward*)
		PArm_BWD : BOOL; (*arm going backward*)
		CapGripper_PICK : BOOL; (*cap gripper is picking*)
	END_STRUCT;
END_TYPE
```

### Program Logical/LogoConvPkg/LogoCOnv (IEC)

#### Main.st - Init, cyclic, exit code
```iecst
PROGRAM _INIT
	(* Insert code here *)
//	 iLogoConv.AOs.LogoConvSpeed:=0.1;
	BasicParameters.Velocity:= 100;
END_PROGRAM

PROGRAM _CYCLIC

	//axis action file
	LogoAxis;

	CASE sLogoConvStep OF
		//waiting for commands
		enWAIT:
			iLogoConv.AOs.LogoConvSpeed:=0;
			IF iLogoConv.Cmd.Start=TRUE THEN
				iLogoConv.Cmd.Start:=FALSE;
				sLogoConvStep:=enOPERATION;
			END_IF;

			//operation mode cap is on
		enOPERATION:

			IF iLogoConv.DIs.LogoConvStart_IR=TRUE THEN
				sLogoConvStep:=enRUNNING;
			END_IF;

			//running the conveyor
		enRUNNING:
			iLogoConv.AOs.LogoConvSpeed:=BasicParameters.Velocity/100;
			IF iLogoConv.DIs.LogoConvExit_IR=TRUE THEN
				sLogoConvStep:=enEXIT;
			END_IF;

			//exit cap from conveyor
		enEXIT:

			IF iLogoConv.Status.Running=FALSE THEN
				sLogoConvStep:=enEXIT;
				//iLogoConv.AOs.LogoConvSpeed:=0;
				sLogoConvStep:=enWAIT;
			END_IF;

			//error mode
		enERROR:
			iLogoConv.AOs.LogoConvSpeed:=0;
			IF iLogoConv.Cmd.ErrorReset=TRUE THEN
				iLogoConv.Cmd.ErrorReset:=FALSE;
				sLogoConvStep:=enWAIT;
			END_IF;
	END_CASE;
END_PROGRAM

PROGRAM _EXIT
	(* Insert code here *)

END_PROGRAM
```

#### Types.typ - Local data types
```iecst
TYPE
	sStep_LogoConv :
		(
		enWAIT,
		enOPERATION,
		enRUNNING,
		enEXIT,
		enERROR
		);
	Step :
		(
		enINITA,
		enSTARTA,
		enPOWER_ONA,
		enHOMEA,
		enOPERATIONA,
		enERRORA
		);
END_TYPE
```

#### Variables.var - Local variables
```iecst
VAR
	iLogoConv : LogoConv_typ;
	sLogoConvStep : sStep_LogoConv;
	BasicParameters : MpAxisBasicParType;
	iFb_MpAxisBasic_0 : MpAxisBasic;
	cmdPower : BOOL;
	cmdHome : BOOL;
	cmdMoveVelocity : BOOL;
	cmdMoveAdditive : BOOL;
	cmdUpdate : BOOL;
	cmdStop : BOOL;
	cmdErrorReset : BOOL;
	iFb_MC_MoveVelocity_0 : MC_MoveVelocity;
	cmdMoveVelocity_ACP10_MC : BOOL;
	strStep : Step;
	ERROR : BOOL;
	iVl_OldVelocity : REAL;
END_VAR
```

#### LogoAxis.st
```iecst
ACTION LogoAxis:

	iFb_MpAxisBasic_0.MpLink := ADR(gAxisBasic);
	iFb_MpAxisBasic_0.Axis := ADR(gAxis01);
	iFb_MpAxisBasic_0.Enable := 1;
	iFb_MpAxisBasic_0.Parameters := ADR(BasicParameters);
	iFb_MpAxisBasic_0();

	//	BasicParameters.Velocity := 1000;
	//	BasicParameters.Distance := 1000;
	//
	IF iVl_OldVelocity<> BasicParameters.Velocity THEN
		iFb_MpAxisBasic_0.Update:=TRUE ;
		IF	iFb_MpAxisBasic_0.UpdateDone=TRUE THEN
			iVl_OldVelocity:= BasicParameters.Velocity;
			iFb_MpAxisBasic_0.Update:=FALSE ;
		END_IF;

	END_IF;
	//	iFb_MC_MoveVelocity_0.Acceleration := 2000;
	//	iFb_MC_MoveVelocity_0.Deceleration := 2000;

	iFb_MC_MoveVelocity_0.Axis := ADR(gAxis01);
	iFb_MpAxisBasic_0.Power := cmdPower;
	iFb_MpAxisBasic_0.Home := cmdHome;
	iFb_MpAxisBasic_0.ErrorReset := cmdErrorReset;
	iFb_MpAxisBasic_0.MoveVelocity := cmdMoveVelocity;
	iFb_MpAxisBasic_0.MoveAdditive;

	//Limit for the torque
	BasicParameters.Torque.Limit:=0.8;

	IF cmdStop=TRUE THEN
		iFb_MpAxisBasic_0.Stop:=TRUE;
		cmdStop:=FALSE;
		IF iFb_MpAxisBasic_0.Stopped=TRUE THEN
			iFb_MpAxisBasic_0.Stop:=FALSE;
		END_IF;
	END_IF;

	IF iFb_MpAxisBasic_0.Error=TRUE THEN
		strStep:=enERRORA;
	END_IF;

	CASE strStep OF

		enINITA:

		enSTARTA:
			IF iFb_MpAxisBasic_0.Info.ReadyToPowerOn = TRUE THEN
				strStep := enPOWER_ONA;
			END_IF
		enPOWER_ONA:
			cmdPower := TRUE;
			IF iFb_MpAxisBasic_0.PowerOn = TRUE THEN
				strStep := enHOMEA;
			END_IF
		enHOMEA:
			cmdHome := TRUE;
			IF iFb_MpAxisBasic_0.IsHomed = TRUE THEN
				strStep := enOPERATIONA;
				cmdHome := FALSE;
			END_IF
		enOPERATIONA:
			IF iFb_MpAxisBasic_0.Error =
				TRUE THEN
				strStep := enERRORA;
			END_IF
			IF cmdMoveAdditive=TRUE THEN
				iFb_MpAxisBasic_0.MoveAdditive:=TRUE;
				cmdMoveAdditive := FALSE;
			END_IF;

		enERRORA:
			cmdPower := FALSE;
			cmdMoveVelocity := FALSE;
			cmdStop := FALSE;
			cmdErrorReset;
			IF iFb_MpAxisBasic_0.Error = FALSE THEN;
				strStep := enSTARTA;
				cmdErrorReset := FALSE;
			END_IF
	END_CASE

	iFb_MpAxisBasic_0();
	iFb_MC_MoveVelocity_0();
END_ACTION
```

#### AlarmsLC.st - not listed in the package file held
```iecst
ACTION AlarmsLC:

	IF iLogoConv.AOs.LogoConvSpeed=0 AND iLogoConv.DIs.LogoConvStart_IR=TRUE THEN
		MpAlarmXSet(gAlarmXCore, 'ConvLogoErr');
		IF MpAlarmXCheckReaction(gAlarmXCore, 'EStop') THEN
		//	iLogoConv.AOs.LogoConvSpeed:=1;
		END_IF
	ELSE
		MpAlarmXReset(gAlarmXCore, 'ConvLogoErr');
	END_IF
END_ACTION
```

### LogoTyp.typ
```iecst
(*Main control for logo conveyor*)

TYPE
	LogoConv_typ : 	STRUCT
		DIs : LogoConvDIs; (*digital inputs*)
		AOs : LogoConvAOs; (*anallog outputs*)
		Cmd : LogoConvCmd; (*commands*)
		Status : LogoConvStatus; (*statuses*)
	END_STRUCT;
END_TYPE

(*Conveyor belt digital inputs*)

TYPE
	LogoConvDIs : 	STRUCT  (*digital inputs*)
		LogoConvStart_IR : BOOL; (*conveyor is started*)
		LogoConvExit_IR : BOOL; (*exiting the conveyor*)
		LogoActPos : REAL; (*actual position of the conveyor belt*)
	END_STRUCT;
END_TYPE

(*analog outputs *)

TYPE
	LogoConvAOs : 	STRUCT  (*analog outputs*)
		LogoConvSpeed : REAL; (*conveyor speed for conveyor*)
	END_STRUCT;
END_TYPE

(*status of the logo conveyor*)

TYPE
	LogoConvStatus : 	STRUCT  (*status for logo conveyor*)
		Running : BOOL; (*running*)
		Error : BOOL; (*in error mode*)
	END_STRUCT;
END_TYPE

(*command to logo conveyor*)

TYPE
	LogoConvCmd : 	STRUCT  (*basic commnds*)
		Start : BOOL; (*stating the conv*)
		Stop : BOOL; (*stopping*)
		Estop : BOOL; (*emergency stop*)
		ErrorReset : BOOL;
	END_STRUCT;
END_TYPE
```

### Program Logical/SortConvPkg/SortConv (IEC)

#### Main.st - Init, cyclic, exit code
```iecst
PROGRAM _INIT
	(* Insert code here *)
	BasicParameters.Velocity:= 100;

END_PROGRAM

PROGRAM _CYCLIC
	(* Insert code here *)
	SortAxisA;
	CASE sSortConvStep OF
		enWAIT:
			IF iSortConv.Cmd.Start=TRUE THEN
				iSortConv.Cmd.Start:=FALSE;
				sSortConvStep:=enOPERATION;
			END_IF;

		enOPERATION:
			iSortConv.Status.Running:=TRUE;
			IF iSortConv.DIs.SortBasicConvStart_IR=TRUE THEN
				iSortConv.AOs.SortBasicConvSpeed:=BasicParameters.Velocity/100;;
				sSortConvStep:=enRUNNING;
			END_IF;

		enRUNNING:
			IF iSortConv.Status.Running=FALSE THEN
				sSortConvStep:=enWAIT;
			END_IF;

		enERROR:
			iSortConv.AOs.SortBasicConvSpeed:=0;
			IF iSortConv.Cmd.ErrorReset=TRUE THEN
				iSortConv.Cmd.ErrorReset:=FALSE;
				sSortConvStep:=enWAIT;
			END_IF;

	END_CASE;
END_PROGRAM

PROGRAM _EXIT
	(* Insert code here *)

END_PROGRAM
```

#### Types.typ - Local data types
```iecst
TYPE
	sStep_SortConv :
		(
		enWAIT,
		enOPERATION,
		enRUNNING,
		enEXIT,
		enERROR,
		enSTOP
		);
	Step :
		(
		enINITA,
		enSTARTA,
		enPOWER_ONA,
		enHOMEA,
		enOPERATIONA,
		enERRORA
		);
END_TYPE
```

#### Variables.var - Local variables
```iecst
VAR
	iSortConv : SortBasicConv_typ;
	sSortConvStep : sStep_SortConv;
	BasicParameters : MpAxisBasicParType;
	iFb_MpAxisBasic_0 : MpAxisBasic;
	cmdPower : BOOL;
	cmdHome : BOOL;
	cmdMoveVelocity : BOOL;
	cmdMoveAdditive : BOOL;
	cmdUpdate : BOOL;
	cmdStop : BOOL;
	cmdErrorReset : BOOL;
	iFb_MC_MoveVelocity_0 : MC_MoveVelocity;
	cmdMoveVelocity_ACP10_MC : BOOL;
	strStep : Step;
	ERROR : BOOL;
END_VAR
```

#### SortAxisA.st
```iecst
ACTION SortAxisA:

	iFb_MpAxisBasic_0.MpLink := ADR(gAxisBasic_1);
	iFb_MpAxisBasic_0.Axis := ADR(gAxis02);
	iFb_MpAxisBasic_0.Enable := 1;
	iFb_MpAxisBasic_0.Parameters := ADR(BasicParameters);
	iFb_MpAxisBasic_0();
//
//	BasicParameters.Velocity := 1000;
//	BasicParameters.Distance := 1000;
//
//	iFb_MC_MoveVelocity_0.Velocity := 1000;
//	iFb_MC_MoveVelocity_0.Acceleration := 2000;
//	iFb_MC_MoveVelocity_0.Deceleration := 2000;

	iFb_MC_MoveVelocity_0.Axis := ADR(gAxis02);
	iFb_MpAxisBasic_0.Power := cmdPower;
	iFb_MpAxisBasic_0.Home := cmdHome;
	iFb_MpAxisBasic_0.ErrorReset := cmdErrorReset;
	iFb_MpAxisBasic_0.MoveVelocity := cmdMoveVelocity;
	iFb_MpAxisBasic_0.MoveAdditive;

	//Limit for the torque
	BasicParameters.Torque.Limit:=0.8;

	IF cmdStop=TRUE THEN
		iFb_MpAxisBasic_0.Stop:=TRUE;
		cmdStop:=FALSE;
		IF iFb_MpAxisBasic_0.Stopped=TRUE THEN
			iFb_MpAxisBasic_0.Stop:=FALSE;
		END_IF;
	END_IF;

	IF iFb_MpAxisBasic_0.Error=TRUE THEN
		strStep:=enERRORA;
	END_IF;

	CASE strStep OF

		enINITA:

		enSTARTA:
			IF iFb_MpAxisBasic_0.Info.ReadyToPowerOn = TRUE THEN
				strStep := enPOWER_ONA;
			END_IF
		enPOWER_ONA:
			cmdPower := TRUE;
			IF iFb_MpAxisBasic_0.PowerOn = TRUE THEN
				strStep := enHOMEA;
			END_IF
		enHOMEA:
			cmdHome := TRUE;
			IF iFb_MpAxisBasic_0.IsHomed = TRUE THEN
				strStep := enOPERATIONA;
				cmdHome := FALSE;
			END_IF
		enOPERATIONA:
			IF iFb_MpAxisBasic_0.Error = TRUE THEN
				strStep := enERRORA;
			END_IF
			IF cmdMoveAdditive=TRUE THEN
				iFb_MpAxisBasic_0.MoveAdditive:=TRUE;
				cmdMoveAdditive := FALSE;
			END_IF;

		enERRORA:
			cmdPower := FALSE;
			cmdMoveVelocity := FALSE;
			cmdStop := FALSE;
			cmdErrorReset;
			IF iFb_MpAxisBasic_0.Error = FALSE THEN;
				strStep := enSTARTA;
				cmdErrorReset := FALSE;
			END_IF
	END_CASE

	iFb_MpAxisBasic_0();
	iFb_MC_MoveVelocity_0();
END_ACTION
```

#### AlarmsSC.st - not listed in the package file held
```iecst
ACTION AlarmsSC:

	IF iSortConv.AOs.SortBasicConvSpeed=0 AND iSortConv.DIs.SortBasicConvStart_IR=TRUE THEN
		MpAlarmXSet(gAlarmXCore, 'ConvSortErr');
		IF MpAlarmXCheckReaction(gAlarmXCore, 'EStop') THEN
			iSortConv.AOs.SortBasicConvSpeed:=1;
		END_IF
	ELSE
		MpAlarmXReset(gAlarmXCore, 'ConvSortErr');
	END_IF
END_ACTION
```

### SortTyp.typ
```iecst
(*Strcutre for main control*)

TYPE
	SortBasicConv_typ : 	STRUCT  (*conveyor main strcutre*)
		DIs : SortBasicConvDIs_typ; (*DI strcture*)
		AOs : SortBasicConvAOs_typ; (*AO strcutre *)
		Status : SortBasicConvStatus_typ; (*status strcuter*)
		Cmd : SortBasicConvCmd_typ; (*commands*)
	END_STRUCT;
END_TYPE

(*Digital outputs*)

TYPE
	SortBasicConvDIs_typ : 	STRUCT  (*sort conveyor Digital inputs*)
		SortBasicConvStart_IR : BOOL; (*IR sesnor detecting*)
	END_STRUCT;
END_TYPE

(*Analog ouputs*)

TYPE
	SortBasicConvAOs_typ : 	STRUCT  (*Analog outputs*)
		SortBasicConvSpeed : REAL; (*conveyor spped of basics*)
	END_STRUCT;
END_TYPE

(*Status for the conv belt'*)

TYPE
	SortBasicConvStatus_typ : 	STRUCT  (*statuses for conveyor*)
		Running : BOOL; (*running mode*)
		Error : BOOL; (*in n errror mode*)
	END_STRUCT;
END_TYPE

(*basic commands*)

TYPE
	SortBasicConvCmd_typ : 	STRUCT  (*basic conveyor command*)
		Start : BOOL; (*starting commadnd*)
		Stop : BOOL; (*stopping*)
		Estop : BOOL; (*emergency stop*)
		ErrorReset : BOOL;
	END_STRUCT;
END_TYPE
```

### Program Logical/ClrDetectPkg/ClrDetect (IEC)

#### Main.st - Init, cyclic, exit code
```iecst
PROGRAM _INIT
	(* Insert code here *)

END_PROGRAM

PROGRAM _CYCLIC
	(* Insert code here *)
	iClrDetect;
	CASE sClrDetectStep OF

		//waiting for start
		enWAIT:
			IF iClrDetect.Cmd.Start=TRUE THEN
				gColorCap:="";
				iClrDetect.Cmd.Start:=FALSE;
				iClrDetect.DOs.CapStopperFWD:=TRUE;
				sClrDetectStep:=enOPERATION;
			END_IF;

			//operation mode if ir detects
		enOPERATION:
			IF iClrDetect.DIs.ColorDetectionIR =TRUE THEN
				sClrDetectStep:=enRUNNING;
			END_IF;

			//running mode
		enRUNNING:
			IF iClrDetect.DIs.ColorDtectMetallic=TRUE THEN
				iClrDetect.Status.iNoOfMetallic:=iClrDetect.Status.iNoOfMetallic+1;
				gColorCap:="Metallic";
				sClrDetectStep:=enEXIT;
			ELSIF iClrDetect.DIs.ColorDtectNotBlack =FALSE AND iClrDetect.DIs.ColorDtectMetallic=FALSE THEN
				iClrDetect.Status.iNoOfBlack:=iClrDetect.Status.iNoOfBlack+1;
				gColorCap:="Black";
				sClrDetectStep:=enEXIT;
			ELSIF iClrDetect.DIs.ColorDtectNotBlack =TRUE AND iClrDetect.DIs.ColorDtectMetallic=FALSE THEN
				iClrDetect.Status.iNoOfRed:=iClrDetect.Status.iNoOfRed+1;
				gColorCap:="RED";
				sClrDetectStep:=enEXIT;
			END_IF;

			//exiting the station
		enEXIT:

			iClrDetect.DOs.CapStopperFWD:=FALSE;
			sClrDetectStep:=enWAIT;

			//error mode
		enERROR:

			iClrDetect.DOs.CapStopperFWD:=TRUE;
			IF iClrDetect.Cmd.ErrorReset=TRUE THEN
				iClrDetect.Cmd.ErrorReset:=FALSE;
				sClrDetectStep:=enWAIT;
			END_IF;

	END_CASE;

END_PROGRAM

PROGRAM _EXIT
	(* Insert code here *)

END_PROGRAM
```

#### Types.typ - Local data types
```iecst
TYPE
	sStep_ClrDetect :
		(
		enWAIT,
		enOPERATION,
		enRUNNING,
		enEXIT,
		enERROR
		);
END_TYPE
```

#### Variables.var - Local variables
```iecst
VAR
	iClrDetect : ClrDetect_typ; (*main color detect strcutre*)
END_VAR
VAR RETAIN
	sClrDetectStep : sStep_ClrDetect;
END_VAR
VAR CONSTANT
	MAXNOCAP : USINT := 9;
END_VAR
```

#### AlarmsCD.st
```iecst
ACTION AlarmsCD:

	IF iClrDetect.Cmd.Estop=TRUE   THEN
		MpAlarmXSet(gAlarmXCore, 'EStopCD');
		iClrDetect.Status.Error:=TRUE;
		IF MpAlarmXCheckReaction(gAlarmXCore, 'EStop') THEN
		//	sClrDetectStep:=enERROR;
		END_IF
	ELSE
		MpAlarmXReset(gAlarmXCore, 'EStopCD');
	END_IF

	IF iClrDetect.Status.iNoOfBlack =MAXNOCAP   OR iClrDetect.Status.iNoOfRed =MAXNOCAP  OR iClrDetect.Status.iNoOfMetallic=MAXNOCAP   THEN
		MpAlarmXSet(gAlarmXCore, 'CapsFull');
		IF MpAlarmXCheckReaction(gAlarmXCore, 'EStop') THEN
			iClrDetect.Status.iNoOfBlack:=0;
			iClrDetect.Status.iNoOfMetallic:=0;
			iClrDetect.Status.iNoOfMetallic:=0;
		END_IF
	ELSE
		MpAlarmXReset(gAlarmXCore, 'CapsFull');
	END_IF
END_ACTION
```

### ClrDetTyp.typ
```iecst
TYPE
	ClrDetect_typ : 	STRUCT  (*main strcuter for colore detection*)
		DIs : DIClrDetect_typ; (*digital inputs*)
		DOs : DOClrDetect_typ; (*digital outputs*)
		Cmd : CmdClrDetect_typ; (*commands*)
		Status : StatusClrDetect_typ; (*status for color*)
	END_STRUCT;
	DIClrDetect_typ : 	STRUCT  (*Digital input strcutuere*)
		ColorDetectionIR : BOOL; (*ir sensor for color detection*)
		ColorDtectNotBlack : BOOL; (*cap is not black*)
		ColorDtectMetallic : BOOL; (*cap is of mettalic color*)
	END_STRUCT;
	DOClrDetect_typ : 	STRUCT  (*do for color detection*)
		CapStopperFWD : BOOL; (*cap stopper in forward direxn*)
	END_STRUCT;
	CmdClrDetect_typ : 	STRUCT  (*color command strcutre*)
		Start : BOOL; (*starting*)
		Stop : BOOL; (*stopping*)
		Estop : BOOL; (*emergency stop pressed*)
		ErrorReset : BOOL;
	END_STRUCT;
	StatusClrDetect_typ : 	STRUCT  (*status for color structure*)
		Running : BOOL; (*running *)
		Error : BOOL; (*error mode*)
		iNoOfRed : USINT;
		iNoOfBlack : USINT;
		iNoOfMetallic : USINT;
	END_STRUCT;
END_TYPE
```

### Program Logical/LaneGatesPkg/LineGates (IEC)

#### Main.st - Init, cyclic, exit code
```iecst
PROGRAM _INIT
	(* Insert code here *)

END_PROGRAM

PROGRAM _CYCLIC
	(* Insert code here *)
	iLineGates;

	CASE sLineGateStep OF
		//waiting for the start
		enWAIT:
			IF iLineGates.Cmd.Start=TRUE THEN
				iLineGates.Cmd.Start:=FALSE;
				iLineGates.Status.Running:=TRUE;
				sLineGateStep:=enOPERATION;
			END_IF;

			//operating the linegagtes
		enOPERATION:
			IF gColorCap="Black" THEN
				iLineGates.DOs.LG1FWD:=TRUE;
				IF iLineGates.DIs.LG1_LFR=TRUE THEN
					sLineGateStep:=enRUNNING;
				END_IF;
			ELSIF gColorCap="Metallic" THEN
				iLineGates.DOs.LW2FWD :=TRUE;
				IF iLineGates.DIs.LG2_LFR=TRUE THEN
					sLineGateStep:=enRUNNING;
				END_IF;
			ELSE
				iLineGates.DOs.LG1FWD:=FALSE;
				iLineGates.DOs.LW2FWD:=FALSE;
				sLineGateStep:=enRUNNING;
			END_IF;

			//running mode
		enRUNNING:

			IF iLineGates.DIs.LaneTopIR=TRUE THEN
				iLineGates.DOs.LG1FWD:=FALSE;
				iLineGates.DOs.LW2FWD:=FALSE;
			END_IF;

			IF iLineGates.DIs.LG1_LBK=TRUE AND  iLineGates.DIs.LG2_LBK=TRUE THEN
				sLineGateStep:=enWAIT;
				iLineGates.Status.Running:=FALSE;
			END_IF;

			//error mode
		enERROR:
			iLineGates.DOs.LG1FWD:=FALSE;
			iLineGates.DOs.LW2FWD:=FALSE;
			IF iLineGates.Cmd.ErrorReset=TRUE THEN
				iLineGates.Cmd.ErrorReset:=FALSE;
				sLineGateStep:=enWAIT;
			END_IF;

	END_CASE;

END_PROGRAM

PROGRAM _EXIT
	(* Insert code here *)

END_PROGRAM
```

#### Types.typ - Local data types
```iecst
TYPE
	sStep_LineGates :
		(
		enWAIT,
		enOPERATION,
		enRUNNING,
		enRESET,
		enEXIT,
		enERROR
		);
END_TYPE
```

#### Variables.var - Local variables
```iecst
VAR
	iLineGates : LineGates_typ; (*main strcuture for line gate*)
	sLineGateStep : sStep_LineGates;
	iNoOfBlack : USINT;
	iNoOfMetallic : USINT;
	iNoOfRed : USINT;
END_VAR
```

#### AlarmsLG.st
```iecst
ACTION AlarmsCD:

	IF iClrDetect.Cmd.Estop=TRUE   THEN
		MpAlarmXSet(gAlarmXCore, 'EStopLG');
		iClrDetect.Status.Error:=TRUE;
		IF MpAlarmXCheckReaction(gAlarmXCore, 'EStop') THEN
			sClrDetectStep:=enERROR;
		END_IF
	ELSE
		MpAlarmXReset(gAlarmXCore, 'EStopLG');
	END_IF

END_ACTION
```

### Types.typ
```iecst
(*main control*)

TYPE
	LineGates_typ : 	STRUCT  (*Line gate main control*)
		Cmd : CmdLineGates_typ; (*command for line gates*)
		Status : StatusLineGates_typ; (*status for line gates*)
		DIs : DILineGates_typ; (*Dis for line gate*)
		DOs : DOLineGates_typ; (*dos for line gates*)
	END_STRUCT;
	DILineGates_typ : 	STRUCT  (*di strcutue for line gate*)
		LG1_LFR : BOOL; (*line gate 1 Left front*)
		LG1_LBK : BOOL; (*line gate 2 Leftback*)
		LG2_LFR : BOOL; (*line gate 1 Left front*)
		LG2_LBK : BOOL; (*line gate 2 Left back*)
		LaneTopIR : BOOL; (*Lane top IR sensor*)
	END_STRUCT;
	DOLineGates_typ : 	STRUCT  (*do line gates*)
		LG1FWD : BOOL; (*lane 1 forward*)
		LW2FWD : BOOL; (*lane 2 forward*)
	END_STRUCT;
	StatusLineGates_typ : 	STRUCT  (*sttus for line gates*)
		Running : BOOL; (*running state*)
		Error : BOOL; (*in errror state*)
	END_STRUCT;
	CmdLineGates_typ : 	STRUCT  (*command to line gates*)
		Start : BOOL; (*starting the line gates*)
		Stop : BOOL; (*stopping the linegate*)
		Estop : BOOL; (*emergency stop for line gate*)
		ErrorReset : BOOL;
	END_STRUCT;
END_TYPE
```

### Program Logical/AutoCtrlPkg/AutoCtrl (IEC)

#### Main.st - Init, cyclic, exit code
```iecst
PROGRAM _INIT
	(* Insert code here *)
	StatusCapPush 		:= PV_xgetadr(ADR('CapPush:iCapPush'),ADR(CapPushAddress),ADR(SizeCapPush));
	StatusPickupArm 	:= PV_xgetadr(ADR('PickupArm:iPickupArm'),ADR(PickupArmAddress),ADR(SizePickupArm));
	StatusLogoCOnv 		:= PV_xgetadr(ADR('LogoCOnv:iLogoConv'),ADR(LogoConvAddress),ADR(SizeLogoConv));
	StatusSortConv		:= PV_xgetadr(ADR('SortConv:iSortConv'), ADR(SortConvAddress), ADR(SizeSortConv));
	StatusClrDetect		:= PV_xgetadr(ADR('ClrDetect:iClrDetect'), ADR(ClrDetectAddress), ADR(SizeClrDetect));
	StatusLineGates		:= PV_xgetadr(ADR('LineGates:iLineGates'), ADR(LineGatesAddress), ADR(SizeLineGates));

	iTimeOut.PT:=T#7s;
END_PROGRAM

PROGRAM _CYCLIC
	(* Insert code here *)
	pCapPush ACCESS CapPushAddress;
	pPickupArm ACCESS PickupArmAddress;
	pLogoConv ACCESS LogoConvAddress;
	pSortConv ACCESS SortConvAddress;
	pClrDetect ACCESS ClrDetectAddress;
	pLineGate ACCESS LineGatesAddress;

	IF iTimeOut.Q=TRUE THEN

	END_IF;
	CASE sAutoStep OF

		//wait state waiting for commmand
		enWAIT:

			IF gMainCmd.Start=TRUE THEN
				gMainCmd.Start:=FALSE;
				sAutoStep:=enSTART;
			END_IF;

			//start state cap is getting pushed
		enSTART:

			pCapPush.Cmd.Start:=TRUE;
			iTimeOut.IN:=TRUE;
			IF pCapPush.Status.Running=TRUE THEN
				sAutoStep:=enCAPPUSH;
				iTimeOut.IN:=FALSE;
			END_IF;

			//cap is pushed
		enCAPPUSH:

			iTimeOut.IN:=TRUE;
			IF pCapPush.DIs.PusherLFR=TRUE THEN
				sAutoStep:=enPICKARM;
				pPickupArm.Cmd.Start:=TRUE;
				iTimeOut.IN:=FALSE;
			END_IF;

			//pick arm picking the cap
		enPICKARM:
			iTimeOut.IN:=TRUE;
			IF pPickupArm.DOs.PArmLBK=TRUE THEN
				pCapPush.DOs.PushFWD:=FALSE;
				sAutoStep:=enLOGOCONV;
				pLogoConv.Cmd.Start:=TRUE;
				iTimeOut.IN:=FALSE;
			END_IF;

			//logo conveyor is on
		enLOGOCONV:
			iTimeOut.IN:=TRUE;
			//IF pLogoConv.DIs.LogoConvExit_IR=TRUE THEN
				IF pLogoConv.DIs.LogoConvExit_IR=TRUE THEN
					sAutoStep:=enSORTCONV;
					pSortConv.Cmd.Start:=TRUE;
					iTimeOut.IN:=FALSE;
				END_IF;
//END_IF;

			//sorting conveyor is on
		enSORTCONV:
				iTimeOut.IN:=TRUE;
				sAutoStep:=enCLRDETECT;
				pClrDetect.Cmd.Start:=TRUE;
				iTimeOut.IN:=FALSE;

			//color detection is on
		enCLRDETECT:
			iTimeOut.IN:=TRUE;

			IF pClrDetect.DOs.CapStopperFWD=FALSE THEN
				sAutoStep:=enLANEGATE;
				pLineGate.Cmd.Start:=TRUE;
				iTimeOut.IN:=FALSE;
			END_IF;

			//lane gate is on
		enLANEGATE:

			iTimeOut.IN:=TRUE;
			IF pLineGate.Status.Running=FALSE THEN
				pSortConv.Status.Running:=FALSE;
				IF pLineGate.Cmd.Stop=TRUE OR pClrDetect.Status.iNoOfBlack=9 OR pClrDetect.Status.iNoOfMetallic=9 OR pClrDetect.Status.iNoOfRed=9 THEN
					iMi_MoveText:="Remove the Cap then only start";
					pLineGate.Cmd.Stop:=FALSE;
					sAutoStep:=enWAIT;
				ELSE
					sAutoStep:=enSTART;
				END_IF;
				iTimeOut.IN:=FALSE;
			END_IF;

	END_CASE;

	iTimeOut();
END_PROGRAM

PROGRAM _EXIT
				(* Insert code here *)

END_PROGRAM
```

#### Types.typ - Local data types
```iecst
TYPE
	Step_AutoCtrl :
		(
		enWAIT,
		enSTART,
		enCAPPUSH,
		enPICKARM,
		enLOGOCONV,
		enSORTCONV,
		enCLRDETECT,
		enLANEGATE,
		enERROR
		);
END_TYPE
```

#### Variables.var - Local variables
```iecst
VAR
	sAutoStep : Step_AutoCtrl;
	StatusCapPush : UINT;
	CapPushAddress : UDINT;
	SizeCapPush : UDINT;
	StatusPickupArm : UINT;
	PickupArmAddress : UDINT;
	SizePickupArm : UDINT;
	StatusLogoCOnv : UINT;
	LogoConvAddress : UDINT;
	SizeLogoConv : UDINT;
	StatusSortConv : UINT;
	SortConvAddress : UDINT;
	SizeSortConv : UDINT;
	StatusClrDetect : UINT;
	ClrDetectAddress : UDINT;
	SizeClrDetect : UDINT;
	StatusLineGates : UINT;
	LineGatesAddress : UDINT;
	SizeLineGates : UDINT;
	pCapPush : REFERENCE TO CapPush_typ;
	pPickupArm : REFERENCE TO PickupArm_typ;
	pLogoConv : REFERENCE TO LogoConv_typ;
	pSortConv : REFERENCE TO SortBasicConv_typ;
	pClrDetect : REFERENCE TO ClrDetect_typ;
	pLineGate : REFERENCE TO LineGates_typ;
	iTimeOut : TON;
	iMi_MoveText : WSTRING[80];
END_VAR
```

#### AutoAlarms.st
```iecst
ACTION AlarmsAuto:

	IF gMainCmd.EStop=TRUE   THEN
		MpAlarmXSet(gAlarmXCore, 'EStopAuto');
		iClrDetect.Status.Error:=TRUE;
		IF MpAlarmXCheckReaction(gAlarmXCore, 'EStop') THEN
			sClrDetectStep:=enERROR;
		END_IF
	ELSE
		MpAlarmXReset(gAlarmXCore, 'EStopAuto');
	END_IF

END_ACTION
```

- Visualisation Logical/mappView (not shown)

Listed in the project but not available here: Logical/acp10etxen, Logical/MNG_Global.typ
